LIN {X 0,Y 186.712,Z 737.862,A -85,B 0,C 180,E1 -23388.136,E2 -23388.136} C_VEL
LIN {X 0,Y 190.106,Z 731.981,A -85,B 0,C 180,E1 -23389.886,E2 -23389.886} C_VEL
LIN {X 0,Y 190.908,Z 730.143,A -85,B 0,C 180,E1 -23390.464,E2 -23390.464} C_VEL
LIN {X 0,Y 192.112,Z 723.011,A -85,B 0,C 180,E1 -23393.119,E2 -23393.119} C_VEL
LIN {X 0,Y 192.536,Z 714.54,A -85,B 0,C 180,E1 -23396.337,E2 -23396.337} C_VEL
LIN {X 0,Y 192.019,Z 709.698,A -85,B 0,C 180,E1 -23398.427,E2 -23398.427} C_VEL
LIN {X 0,Y 189.959,Z 701.617,A -85,B 0,C 180,E1 -23402.676,E2 -23402.676} C_VEL
LIN {X 0,Y 188.484,Z 698.004,A -85,B 0,C 180,E1 -23405.153,E2 -23405.153} C_VEL
LIN {X 0,Y 186.546,Z 693.819,A -85,B 0,C 180,E1 -23408.667,E2 -23408.667} C_VEL
LIN {X 0,Y 184.642,Z 689.744,A -85,B 0,C 180,E1 -23413.201,E2 -23413.201} C_VEL
LIN {X 0,Y 183.126,Z 688.308,A -85,B 0,C 180,E1 -23417.88,E2 -23417.88} C_VEL
LIN {X 0,Y 182.793,Z 688.035,A -85,B 0,C 180,E1 -23422.672,E2 -23422.672} C_VEL
LIN {X 0,Y 183.551,Z 689.151,A -85,B 0,C 180,E1 -23427.353,E2 -23427.353} C_VEL
LIN {X 0,Y 184.381,Z 690.199,A -85,B 0,C 180,E1 -23429.704,E2 -23429.704} C_VEL
LIN {X 0,Y 185.28,Z 692.119,A -85,B 0,C 180,E1 -23432.076,E2 -23432.076} C_VEL
LIN {X 0,Y 186.909,Z 695.318,A -85,B 0,C 180,E1 -23435.291,E2 -23435.291} C_VEL
LIN {X 0,Y 189.282,Z 700.42,A -85,B 0,C 180,E1 -23439.139,E2 -23439.139} C_VEL
LIN {X 0,Y 191.326,Z 707.048,A -85,B 0,C 180,E1 -23442.723,E2 -23442.723} C_VEL
LIN {X 0,Y 192.053,Z 709.901,A -85,B 0,C 180,E1 -23444.05,E2 -23444.05} C_VEL
LIN {X 0,Y 192.147,Z 713.982,A -85,B 0,C 180,E1 -23445.498,E2 -23445.498} C_VEL
LIN {X 0,Y 191.189,Z 723.676,A -85,B 0,C 180,E1 -23448.574,E2 -23448.574} C_VEL
LIN {X 0,Y 189.395,Z 732.577,A -85,B 0,C 180,E1 -23451.427,E2 -23451.427} C_VEL
LIN {X 0,Y 186.775,Z 741.156,A -85,B 0,C 180,E1 -23454.323,E2 -23454.323} C_VEL
LIN {X 0,Y 184.598,Z 745.61,A -85,B 0,C 180,E1 -23455.838,E2 -23455.838} C_VEL
LIN {X 0,Y 179.665,Z 753.449,A -85,B 0,C 180,E1 -23458.783,E2 -23458.783} C_VEL
LIN {X 0,Y 174.569,Z 760.74,A -85,B 0,C 180,E1 -23462.338,E2 -23462.338} C_VEL
LIN {X 0,Y 170.932,Z 765.844,A -85,B 0,C 180,E1 -23465.724,E2 -23465.724} C_VEL
LIN {X 0,Y 167.819,Z 769.773,A -85,B 0,C 180,E1 -23469.148,E2 -23469.148} C_VEL
LIN {X 0,Y 165.259,Z 772.729,A -85,B 0,C 180,E1 -23472.682,E2 -23472.682} C_VEL
LIN {X 0,Y 163.137,Z 775.246,A -85,B 0,C 180,E1 -23477.562,E2 -23477.562} C_VEL
LIN {X 0,Y 162.025,Z 776.252,A -85,B 0,C 180,E1 -23482.524,E2 -23482.524} C_VEL
LIN {X 0,Y 161.851,Z 775.794,A -85,B 0,C 180,E1 -23487.106,E2 -23487.106} C_VEL
LIN {X 0,Y 161.904,Z 775.442,A -85,B 0,C 180,E1 -23488.77,E2 -23488.77} C_VEL
LIN {X 0,Y 162.003,Z 776.041,A -85,B 0,C 180,E1 -23490.001,E2 -23490.001} C_VEL
LIN {X 0,Y 161.833,Z 777.013,A -85,B 0,C 180,E1 -23492.77,E2 -23492.77} C_VEL
LIN {X 0,Y 162.035,Z 777.558,A -85,B 0,C 180,E1 -23497.478,E2 -23497.478} C_VEL
LIN {X 0,Y 163.149,Z 776.604,A -85,B 0,C 180,E1 -23502.439,E2 -23502.439} C_VEL
LIN {X 0,Y 163.38,Z 776.322,A -85,B 0,C 180,E1 -23503.114,E2 -23503.114} C_VEL
LIN {X 0,Y 163.558,Z 775.484,A -85,B 0,C 180,E1 -23505.161,E2 -23505.161} C_VEL
LIN {X 0,Y 162.556,Z 773.609,A -85,B 0,C 180,E1 -23508.569,E2 -23508.569} C_VEL
LIN {X 0,Y 162.155,Z 771.222,A -85,B 0,C 180,E1 -23511.955,E2 -23511.955} C_VEL
LIN {X 0,Y 163.246,Z 769.393,A -85,B 0,C 180,E1 -23513.891,E2 -23513.891} C_VEL
LIN {X 0,Y 167.46,Z 764.248,A -85,B 0,C 180,E1 -23517.989,E2 -23517.989} C_VEL
LIN {X 0,Y 172.073,Z 758.395,A -85,B 0,C 180,E1 -23521.384,E2 -23521.384} C_VEL
LIN {X 0,Y 177.108,Z 751.485,A -85,B 0,C 180,E1 -23524.436,E2 -23524.436} C_VEL
LIN {X 0,Y 180.696,Z 746.067,A -85,B 0,C 180,E1 -23526.381,E2 -23526.381} C_VEL
LIN {X 0,Y 183.191,Z 739.813,A -85,B 0,C 180,E1 -23528.764,E2 -23528.764} C_VEL
LIN {X 0,Y 185.082,Z 732.261,A -85,B 0,C 180,E1 -23531.646,E2 -23531.646} C_VEL
LIN {X 0,Y 186.028,Z 725.848,A -85,B 0,C 180,E1 -23534.126,E2 -23534.126} C_VEL
LIN {X 0,Y 186.099,Z 721.842,A -85,B 0,C 180,E1 -23535.852,E2 -23535.852} C_VEL
LIN {X 0,Y 185.417,Z 716.956,A -85,B 0,C 180,E1 -23538.448,E2 -23538.448} C_VEL
LIN {X 0,Y 183.96,Z 710.944,A -85,B 0,C 180,E1 -23542.319,E2 -23542.319} C_VEL
LIN {X 0,Y 183.024,Z 707.744,A -85,B 0,C 180,E1 -23544.831,E2 -23544.831} C_VEL
LIN {X 0,Y 181.454,Z 703.142,A -85,B 0,C 180,E1 -23549.767,E2 -23549.767} C_VEL
LIN {X 0,Y 181.071,Z 701.312,A -85,B 0,C 180,E1 -23552.24,E2 -23552.24} C_VEL
LIN {X 0,Y 180.413,Z 699.995,A -85,B 0,C 180,E1 -23557.074,E2 -23557.074} C_VEL
LIN {X 0,Y 180.881,Z 699.879,A -85,B 0,C 180,E1 -23561.891,E2 -23561.891} C_VEL
LIN {X 0,Y 181.587,Z 700.232,A -85,B 0,C 180,E1 -23564.281,E2 -23564.281} C_VEL
LIN {X 0,Y 182.735,Z 703.422,A -85,B 0,C 180,E1 -23568.913,E2 -23568.913} C_VEL
LIN {X 0,Y 183.638,Z 705.359,A -85,B 0,C 180,E1 -23571.194,E2 -23571.194} C_VEL
LIN {X 0,Y 185.128,Z 709.014,A -85,B 0,C 180,E1 -23574.554,E2 -23574.554} C_VEL
LIN {X 0,Y 186.172,Z 712.751,A -85,B 0,C 180,E1 -23577.188,E2 -23577.188} C_VEL
LIN {X 0,Y 187.119,Z 718.537,A -85,B 0,C 180,E1 -23580.538,E2 -23580.538} C_VEL
LIN {X 0,Y 187.078,Z 723.111,A -85,B 0,C 180,E1 -23582.692,E2 -23582.692} C_VEL
LIN {X 0,Y 186.215,Z 730.51,A -85,B 0,C 180,E1 -23585.957,E2 -23585.957} C_VEL
LIN {X 0,Y 185.472,Z 733.89,A -85,B 0,C 180,E1 -23587.406,E2 -23587.406} C_VEL
LIN {X 0,Y 182.996,Z 738.287,A -85,B 0,C 180,E1 -23588.837,E2 -23588.837} C_VEL
LIN {X 0,Y 177.113,Z 746.781,A -85,B 0,C 180,E1 -23592.017,E2 -23592.017} C_VEL
LIN {X 0,Y 171.766,Z 753.637,A -85,B 0,C 180,E1 -23595.424,E2 -23595.424} C_VEL
LIN {X 0,Y 167.943,Z 758.159,A -85,B 0,C 180,E1 -23598.405,E2 -23598.405} C_VEL
LIN {X 0,Y 164.43,Z 761.942,A -85,B 0,C 180,E1 -23601.652,E2 -23601.652} C_VEL
LIN {X 0,Y 160.739,Z 765.467,A -85,B 0,C 180,E1 -23605.927,E2 -23605.927} C_VEL
LIN {X 0,Y 158.579,Z 767.219,A -85,B 0,C 180,E1 -23609.177,E2 -23609.177} C_VEL
LIN {X 0,Y 156.907,Z 768.33,A -85,B 0,C 180,E1 -23612.513,E2 -23612.513} C_VEL
LIN {X 0,Y 155.638,Z 768.732,A -85,B 0,C 180,E1 -23615.947,E2 -23615.947} C_VEL
LIN {X 0,Y 154.834,Z 768.465,A -85,B 0,C 180,E1 -23619.497,E2 -23619.497} C_VEL
LIN {X 0,Y 154.381,Z 767.416,A -85,B 0,C 180,E1 -23623.248,E2 -23623.248} C_VEL
LIN {X 0,Y 154.361,Z 765.565,A -85,B 0,C 180,E1 -23626.925,E2 -23626.925} C_VEL
LIN {X 0,Y 154.778,Z 762.954,A -85,B 0,C 180,E1 -23630.527,E2 -23630.527} C_VEL
LIN {X 0,Y 155.489,Z 759.109,A -85,B 0,C 180,E1 -23634.448,E2 -23634.448} C_VEL
LIN {X 0,Y 156.66,Z 753.93,A -85,B 0,C 180,E1 -23638.471,E2 -23638.471} C_VEL
LIN {X 0,Y 158.448,Z 747.231,A -85,B 0,C 180,E1 -23642.512,E2 -23642.512} C_VEL
LIN {X 0,Y 160.896,Z 738.567,A -85,B 0,C 180,E1 -23646.533,E2 -23646.533} C_VEL
LIN {X 0,Y 163.527,Z 729.361,A -85,B 0,C 180,E1 -23649.889,E2 -23649.889} C_VEL
LIN {X 0,Y 166.295,Z 719.218,A -85,B 0,C 180,E1 -23652.791,E2 -23652.791} C_VEL
LIN {X 0,Y 167.408,Z 714.851,A -85,B 0,C 180,E1 -23653.851,E2 -23653.851} C_VEL
LIN {X 0,Y 166.812,Z 706.424,A -85,B 0,C 180,E1 -23655.978,E2 -23655.978} C_VEL
LIN {X 0,Y 165.34,Z 695.499,A -85,B 0,C 180,E1 -23658.413,E2 -23658.413} C_VEL
LIN {X 0,Y 163.12,Z 683.74,A -85,B 0,C 180,E1 -23660.701,E2 -23660.701} C_VEL
LIN {X 0,Y 159.913,Z 670.534,A -85,B 0,C 180,E1 -23662.899,E2 -23662.899} C_VEL
LIN {X 0,Y 158.501,Z 667.234,A -85,B 0,C 180,E1 -23663.475,E2 -23663.475} C_VEL
LIN {X 0,Y 157.726,Z 664.838,A -85,B 0,C 180,E1 -23663.924,E2 -23663.924} C_VEL
LIN {X 0,Y 158.258,Z 664.771,A -85,B 0,C 180,E1 -23669.999,E2 -23669.999} C_VEL
LIN {X 0,Y 157.677,Z 664.846,A -85,B 0,C 180,E1 -23675.354,E2 -23675.354} C_VEL
LIN {X 0,Y 158.763,Z 667.875,A -85,B 0,C 180,E1 -23675.874,E2 -23675.874} C_VEL
LIN {X 0,Y 162.128,Z 676.352,A -85,B 0,C 180,E1 -23677.393,E2 -23677.393} C_VEL
LIN {X 0,Y 164.537,Z 688.841,A -85,B 0,C 180,E1 -23679.554,E2 -23679.554} C_VEL
LIN {X 0,Y 166.157,Z 699.914,A -85,B 0,C 180,E1 -23681.804,E2 -23681.804} C_VEL
LIN {X 0,Y 167.206,Z 710.54,A -85,B 0,C 180,E1 -23684.295,E2 -23684.295} C_VEL
LIN {X 0,Y 167.459,Z 713.795,A -85,B 0,C 180,E1 -23685.143,E2 -23685.143} C_VEL
LIN {X 0,Y 164.601,Z 724.758,A -85,B 0,C 180,E1 -23687.961,E2 -23687.961} C_VEL
LIN {X 0,Y 162.062,Z 733.921,A -85,B 0,C 180,E1 -23690.962,E2 -23690.962} C_VEL
LIN {X 0,Y 159.416,Z 743.059,A -85,B 0,C 180,E1 -23694.759,E2 -23694.759} C_VEL
LIN {X 0,Y 157.616,Z 749.693,A -85,B 0,C 180,E1 -23698.256,E2 -23698.256} C_VEL
LIN {X 0,Y 156.377,Z 754.45,A -85,B 0,C 180,E1 -23701.36,E2 -23701.36} C_VEL
LIN {X 0,Y 155.235,Z 759.42,A -85,B 0,C 180,E1 -23705.42,E2 -23705.42} C_VEL
LIN {X 0,Y 154.449,Z 763.205,A -85,B 0,C 180,E1 -23709.571,E2 -23709.571} C_VEL
LIN {X 0,Y 154.222,Z 765.534,A -85,B 0,C 180,E1 -23713.186,E2 -23713.186} C_VEL
LIN {X 0,Y 154.357,Z 767.123,A -85,B 0,C 180,E1 -23716.924,E2 -23716.924} C_VEL
LIN {X 0,Y 154.91,Z 767.907,A -85,B 0,C 180,E1 -23720.568,E2 -23720.568} C_VEL
LIN {X 0,Y 155.925,Z 767.942,A -85,B 0,C 180,E1 -23724.222,E2 -23724.222} C_VEL
LIN {X 0,Y 157.494,Z 767.132,A -85,B 0,C 180,E1 -23727.976,E2 -23727.976} C_VEL
LIN {X 0,Y 159.633,Z 765.454,A -85,B 0,C 180,E1 -23731.702,E2 -23731.702} C_VEL
LIN {X 0,Y 162.394,Z 762.886,A -85,B 0,C 180,E1 -23735.341,E2 -23735.341} C_VEL
LIN {X 0,Y 165.753,Z 759.343,A -85,B 0,C 180,E1 -23738.874,E2 -23738.874} C_VEL
LIN {X 0,Y 169.733,Z 754.752,A -85,B 0,C 180,E1 -23742.235,E2 -23742.235} C_VEL
LIN {X 0,Y 174.266,Z 748.995,A -85,B 0,C 180,E1 -23745.438,E2 -23745.438} C_VEL
LIN {X 0,Y 179.772,Z 741.207,A -85,B 0,C 180,E1 -23748.728,E2 -23748.728} C_VEL
LIN {X 0,Y 184.839,Z 733.12,A -85,B 0,C 180,E1 -23751.323,E2 -23751.323} C_VEL
LIN {X 0,Y 185.992,Z 729.01,A -85,B 0,C 180,E1 -23752.913,E2 -23752.913} C_VEL
LIN {X 0,Y 187.104,Z 722.14,A -85,B 0,C 180,E1 -23755.692,E2 -23755.692} C_VEL
LIN {X 0,Y 187.392,Z 716.951,A -85,B 0,C 180,E1 -23757.851,E2 -23757.851} C_VEL
LIN {X 0,Y 186.623,Z 711.316,A -85,B 0,C 180,E1 -23760.783,E2 -23760.783} C_VEL
LIN {X 0,Y 185.786,Z 707.026,A -85,B 0,C 180,E1 -23763.253,E2 -23763.253} C_VEL
LIN {X 0,Y 184.533,Z 703.526,A -85,B 0,C 180,E1 -23765.839,E2 -23765.839} C_VEL
LIN {X 0,Y 183.23,Z 700.177,A -85,B 0,C 180,E1 -23768.825,E2 -23768.825} C_VEL
LIN {X 0,Y 181.68,Z 696.213,A -85,B 0,C 180,E1 -23773.421,E2 -23773.421} C_VEL
LIN {X 0,Y 180.353,Z 694.814,A -85,B 0,C 180,E1 -23778.164,E2 -23778.164} C_VEL
LIN {X 0,Y 180.118,Z 694.644,A -85,B 0,C 180,E1 -23782.966,E2 -23782.966} C_VEL
LIN {X 0,Y 180.917,Z 695.911,A -85,B 0,C 180,E1 -23787.785,E2 -23787.785} C_VEL
LIN {X 0,Y 181.693,Z 697.21,A -85,B 0,C 180,E1 -23790.189,E2 -23790.189} C_VEL
LIN {X 0,Y 183.599,Z 701.621,A -85,B 0,C 180,E1 -23795.043,E2 -23795.043} C_VEL
LIN {X 0,Y 185.399,Z 706.086,A -85,B 0,C 180,E1 -23798.583,E2 -23798.583} C_VEL
LIN {X 0,Y 187.123,Z 713.019,A -85,B 0,C 180,E1 -23802.536,E2 -23802.536} C_VEL
LIN {X 0,Y 187.343,Z 716.031,A -85,B 0,C 180,E1 -23803.859,E2 -23803.859} C_VEL
LIN {X 0,Y 186.21,Z 724.617,A -85,B 0,C 180,E1 -23806.804,E2 -23806.804} C_VEL
LIN {X 0,Y 184.276,Z 733.14,A -85,B 0,C 180,E1 -23809.709,E2 -23809.709} C_VEL
LIN {X 0,Y 181.73,Z 740.888,A -85,B 0,C 180,E1 -23812.477,E2 -23812.477} C_VEL
LIN {X 0,Y 179.722,Z 745.256,A -85,B 0,C 180,E1 -23814.087,E2 -23814.087} C_VEL
LIN {X 0,Y 174.506,Z 753.117,A -85,B 0,C 180,E1 -23817.066,E2 -23817.066} C_VEL
LIN {X 0,Y 169.726,Z 759.549,A -85,B 0,C 180,E1 -23820.207,E2 -23820.207} C_VEL
LIN {X 0,Y 165.66,Z 764.734,A -85,B 0,C 180,E1 -23823.549,E2 -23823.549} C_VEL
LIN {X 0,Y 162.274,Z 768.848,A -85,B 0,C 180,E1 -23827.06,E2 -23827.06} C_VEL
LIN {X 0,Y 160.211,Z 771.067,A -85,B 0,C 180,E1 -23829.457,E2 -23829.457} C_VEL
LIN {X 0,Y 158.477,Z 772.835,A -85,B 0,C 180,E1 -23831.916,E2 -23831.916} C_VEL
LIN {X 0,Y 156.187,Z 775.195,A -85,B 0,C 180,E1 -23836.999,E2 -23836.999} C_VEL
LIN {X 0,Y 155.443,Z 775.823,A -85,B 0,C 180,E1 -23839.582,E2 -23839.582} C_VEL
LIN {X 0,Y 154.971,Z 776.051,A -85,B 0,C 180,E1 -23842.182,E2 -23842.182} C_VEL
LIN {X 0,Y 154.783,Z 775.877,A -85,B 0,C 180,E1 -23844.791,E2 -23844.791} C_VEL
LIN {X 0,Y 154.831,Z 774.955,A -85,B 0,C 180,E1 -23848.697,E2 -23848.697} C_VEL
LIN {X 0,Y 154.91,Z 775.623,A -85,B 0,C 180,E1 -23850.001,E2 -23850.001} C_VEL
LIN {X 0,Y 154.746,Z 776.569,A -85,B 0,C 180,E1 -23852.604,E2 -23852.604} C_VEL
LIN {X 0,Y 154.781,Z 777.133,A -85,B 0,C 180,E1 -23855.211,E2 -23855.211} C_VEL
LIN {X 0,Y 155.456,Z 777.136,A -85,B 0,C 180,E1 -23860.42,E2 -23860.42} C_VEL
LIN {X 0,Y 157.208,Z 775.581,A -85,B 0,C 180,E1 -23865.56,E2 -23865.56} C_VEL
LIN {X 0,Y 160.266,Z 772.531,A -85,B 0,C 180,E1 -23870.538,E2 -23870.538} C_VEL
LIN {X 0,Y 163.246,Z 769.393,A -85,B 0,C 180,E1 -23873.891,E2 -23873.891} C_VEL
LIN {X 0,Y 163.829,Z 768.103,A -85,B 0,C 180,E1 -23875.198,E2 -23875.198} C_VEL
LIN {X 0,Y 163.133,Z 766.066,A -85,B 0,C 180,E1 -23877.448,E2 -23877.448} C_VEL
LIN {X 0,Y 162.649,Z 763.801,A -85,B 0,C 180,E1 -23879.682,E2 -23879.682} C_VEL
LIN {X 0,Y 163.534,Z 762.125,A -85,B 0,C 180,E1 -23880.914,E2 -23880.914} C_VEL
LIN {X 0,Y 168.641,Z 755.959,A -85,B 0,C 180,E1 -23884.237,E2 -23884.237} C_VEL
LIN {X 0,Y 174.162,Z 748.613,A -85,B 0,C 180,E1 -23887.251,E2 -23887.251} C_VEL
LIN {X 0,Y 175.79,Z 745.856,A -85,B 0,C 180,E1 -23888.294,E2 -23888.294} C_VEL
LIN {X 0,Y 178.272,Z 739.539,A -85,B 0,C 180,E1 -23890.899,E2 -23890.899} C_VEL
LIN {X 0,Y 180.181,Z 732.465,A -85,B 0,C 180,E1 -23893.817,E2 -23893.817} C_VEL
LIN {X 0,Y 180.864,Z 728.249,A -85,B 0,C 180,E1 -23895.618,E2 -23895.618} C_VEL
LIN {X 0,Y 180.912,Z 724.418,A -85,B 0,C 180,E1 -23897.571,E2 -23897.571} C_VEL
LIN {X 0,Y 180.434,Z 720.331,A -85,B 0,C 180,E1 -23900.009,E2 -23900.009} C_VEL
LIN {X 0,Y 179.734,Z 716.555,A -85,B 0,C 180,E1 -23902.702,E2 -23902.702} C_VEL
LIN {X 0,Y 178.671,Z 712.164,A -85,B 0,C 180,E1 -23906.586,E2 -23906.586} C_VEL
LIN {X 0,Y 177.698,Z 708.058,A -85,B 0,C 180,E1 -23911.667,E2 -23911.667} C_VEL
LIN {X 0,Y 177.351,Z 706.922,A -85,B 0,C 180,E1 -23914.157,E2 -23914.157} C_VEL
LIN {X 0,Y 177.183,Z 706.121,A -85,B 0,C 180,E1 -23919.085,E2 -23919.085} C_VEL
LIN {X 0,Y 178.103,Z 706.432,A -85,B 0,C 180,E1 -23923.965,E2 -23923.965} C_VEL
LIN {X 0,Y 179.061,Z 709.599,A -85,B 0,C 180,E1 -23928.884,E2 -23928.884} C_VEL
LIN {X 0,Y 180.21,Z 712.8,A -85,B 0,C 180,E1 -23932.516,E2 -23932.516} C_VEL
LIN {X 0,Y 181.234,Z 716.246,A -85,B 0,C 180,E1 -23935.552,E2 -23935.552} C_VEL
LIN {X 0,Y 181.903,Z 721.342,A -85,B 0,C 180,E1 -23938.893,E2 -23938.893} C_VEL
LIN {X 0,Y 181.891,Z 725.332,A -85,B 0,C 180,E1 -23941.107,E2 -23941.107} C_VEL
LIN {X 0,Y 180.818,Z 732.308,A -85,B 0,C 180,E1 -23944.459,E2 -23944.459} C_VEL
LIN {X 0,Y 179.859,Z 735.959,A -85,B 0,C 180,E1 -23946.169,E2 -23946.169} C_VEL
LIN {X 0,Y 175.815,Z 742.199,A -85,B 0,C 180,E1 -23948.322,E2 -23948.322} C_VEL
LIN {X 0,Y 170.597,Z 749.046,A -85,B 0,C 180,E1 -23951.171,E2 -23951.171} C_VEL
LIN {X 0,Y 164.883,Z 755.647,A -85,B 0,C 180,E1 -23954.818,E2 -23954.818} C_VEL
LIN {X 0,Y 161.094,Z 759.676,A -85,B 0,C 180,E1 -23957.782,E2 -23957.782} C_VEL
LIN {X 0,Y 156.181,Z 764.286,A -85,B 0,C 180,E1 -23962.488,E2 -23962.488} C_VEL
LIN {X 0,Y 152.389,Z 767.295,A -85,B 0,C 180,E1 -23967.464,E2 -23967.464} C_VEL
LIN {X 0,Y 149.789,Z 768.73,A -85,B 0,C 180,E1 -23972.375,E2 -23972.375} C_VEL
LIN {X 0,Y 147.973,Z 768.797,A -85,B 0,C 180,E1 -23978.129,E2 -23978.129} C_VEL
LIN {X 0,Y 147.393,Z 767.88,A -85,B 0,C 180,E1 -23981.879,E2 -23981.879} C_VEL
LIN {X 0,Y 147.228,Z 766.194,A -85,B 0,C 180,E1 -23985.728,E2 -23985.728} C_VEL
LIN {X 0,Y 147.553,Z 763.649,A -85,B 0,C 180,E1 -23989.649,E2 -23989.649} C_VEL
LIN {X 0,Y 148.227,Z 760.03,A -85,B 0,C 180,E1 -23993.711,E2 -23993.711} C_VEL
LIN {X 0,Y 149.324,Z 755.089,A -85,B 0,C 180,E1 -23997.907,E2 -23997.907} C_VEL
LIN {X 0,Y 151.082,Z 748.412,A -85,B 0,C 180,E1 -24002.277,E2 -24002.277} C_VEL
LIN {X 0,Y 153.473,Z 740.442,A -85,B 0,C 180,E1 -24006.329,E2 -24006.329} C_VEL
LIN {X 0,Y 155.942,Z 731.984,A -85,B 0,C 180,E1 -24009.701,E2 -24009.701} C_VEL
LIN {X 0,Y 158.943,Z 721.609,A -85,B 0,C 180,E1 -24012.966,E2 -24012.966} C_VEL
LIN {X 0,Y 160.628,Z 714.624,A -85,B 0,C 180,E1 -24014.779,E2 -24014.779} C_VEL
LIN {X 0,Y 159.59,Z 703.661,A -85,B 0,C 180,E1 -24017.634,E2 -24017.634} C_VEL
LIN {X 0,Y 158.012,Z 692.808,A -85,B 0,C 180,E1 -24020.075,E2 -24020.075} C_VEL
LIN {X 0,Y 155.855,Z 681.966,A -85,B 0,C 180,E1 -24022.224,E2 -24022.224} C_VEL
LIN {X 0,Y 153.244,Z 671.76,A -85,B 0,C 180,E1 -24024.035,E2 -24024.035} C_VEL
LIN {X 0,Y 150.838,Z 666.576,A -85,B 0,C 180,E1 -24025.071,E2 -24025.071} C_VEL
LIN {X 0,Y 150.7,Z 665.712,A -85,B 0,C 180,E1 -24025.318,E2 -24025.318} C_VEL
LIN {X 0,Y 151.218,Z 665.648,A -85,B 0,C 180,E1 -24029.999,E2 -24029.999} C_VEL
LIN {X 0,Y 150.738,Z 665.905,A -85,B 0,C 180,E1 -24034.093,E2 -24034.093} C_VEL
LIN {X 0,Y 151.813,Z 668.79,A -85,B 0,C 180,E1 -24034.604,E2 -24034.604} C_VEL
LIN {X 0,Y 155.865,Z 678.865,A -85,B 0,C 180,E1 -24036.595,E2 -24036.595} C_VEL
LIN {X 0,Y 158.207,Z 691.938,A -85,B 0,C 180,E1 -24039.049,E2 -24039.049} C_VEL
LIN {X 0,Y 159.66,Z 702.785,A -85,B 0,C 180,E1 -24041.424,E2 -24041.424} C_VEL
LIN {X 0,Y 160.566,Z 713.802,A -85,B 0,C 180,E1 -24044.252,E2 -24044.252} C_VEL
LIN {X 0,Y 159.327,Z 719.367,A -85,B 0,C 180,E1 -24045.674,E2 -24045.674} C_VEL
LIN {X 0,Y 156.522,Z 729.436,A -85,B 0,C 180,E1 -24048.688,E2 -24048.688} C_VEL
LIN {X 0,Y 153.859,Z 738.321,A -85,B 0,C 180,E1 -24052.069,E2 -24052.069} C_VEL
LIN {X 0,Y 151.448,Z 746.582,A -85,B 0,C 180,E1 -24056.073,E2 -24056.073} C_VEL
LIN {X 0,Y 149.589,Z 753.402,A -85,B 0,C 180,E1 -24060.334,E2 -24060.334} C_VEL
LIN {X 0,Y 148.276,Z 758.714,A -85,B 0,C 180,E1 -24064.663,E2 -24064.663} C_VEL
LIN {X 0,Y 147.544,Z 762.128,A -85,B 0,C 180,E1 -24068.258,E2 -24068.258} C_VEL
LIN {X 0,Y 147.155,Z 764.792,A -85,B 0,C 180,E1 -24071.96,E2 -24071.96} C_VEL
LIN {X 0,Y 147.167,Z 766.685,A -85,B 0,C 180,E1 -24075.75,E2 -24075.75} C_VEL
LIN {X 0,Y 147.609,Z 767.842,A -85,B 0,C 180,E1 -24079.621,E2 -24079.621} C_VEL
LIN {X 0,Y 148.545,Z 768.228,A -85,B 0,C 180,E1 -24083.541,E2 -24083.541} C_VEL
LIN {X 0,Y 150.064,Z 767.811,A -85,B 0,C 180,E1 -24087.456,E2 -24087.456} C_VEL
LIN {X 0,Y 152.986,Z 765.888,A -85,B 0,C 180,E1 -24092.652,E2 -24092.652} C_VEL
LIN {X 0,Y 156.974,Z 762.504,A -85,B 0,C 180,E1 -24097.553,E2 -24097.553} C_VEL
LIN {X 0,Y 160.383,Z 759.155,A -85,B 0,C 180,E1 -24100.813,E2 -24100.813} C_VEL
LIN {X 0,Y 165.186,Z 753.943,A -85,B 0,C 180,E1 -24104.579,E2 -24104.579} C_VEL
LIN {X 0,Y 170.697,Z 747.199,A -85,B 0,C 180,E1 -24108.12,E2 -24108.12} C_VEL
LIN {X 0,Y 176.788,Z 738.848,A -85,B 0,C 180,E1 -24111.387,E2 -24111.387} C_VEL
LIN {X 0,Y 179.162,Z 735.261,A -85,B 0,C 180,E1 -24112.534,E2 -24112.534} C_VEL
LIN {X 0,Y 180.694,Z 730.715,A -85,B 0,C 180,E1 -24114.42,E2 -24114.42} C_VEL
LIN {X 0,Y 182.125,Z 723.016,A -85,B 0,C 180,E1 -24117.788,E2 -24117.788} C_VEL
LIN {X 0,Y 182.269,Z 719.618,A -85,B 0,C 180,E1 -24119.448,E2 -24119.448} C_VEL
LIN {X 0,Y 181.493,Z 713.117,A -85,B 0,C 180,E1 -24123.33,E2 -24123.33} C_VEL
LIN {X 0,Y 181.206,Z 711.44,A -85,B 0,C 180,E1 -24124.449,E2 -24124.449} C_VEL
LIN {X 0,Y 179.582,Z 706.307,A -85,B 0,C 180,E1 -24129.006,E2 -24129.006} C_VEL
LIN {X 0,Y 178.367,Z 702.486,A -85,B 0,C 180,E1 -24133.675,E2 -24133.675} C_VEL
LIN {X 0,Y 177.249,Z 701.19,A -85,B 0,C 180,E1 -24138.494,E2 -24138.494} C_VEL
LIN {X 0,Y 177.115,Z 701.141,A -85,B 0,C 180,E1 -24143.379,E2 -24143.379} C_VEL
LIN {X 0,Y 177.425,Z 701.664,A -85,B 0,C 180,E1 -24145.831,E2 -24145.831} C_VEL
LIN {X 0,Y 178.435,Z 703.477,A -85,B 0,C 180,E1 -24149.947,E2 -24149.947} C_VEL
LIN {X 0,Y 180.047,Z 707.893,A -85,B 0,C 180,E1 -24154.946,E2 -24154.946} C_VEL
LIN {X 0,Y 181.359,Z 712.066,A -85,B 0,C 180,E1 -24158.318,E2 -24158.318} C_VEL
LIN {X 0,Y 182.374,Z 717.42,A -85,B 0,C 180,E1 -24161.588,E2 -24161.588} C_VEL
LIN {X 0,Y 182.406,Z 720.274,A -85,B 0,C 180,E1 -24162.942,E2 -24162.942} C_VEL
LIN {X 0,Y 180.99,Z 727.677,A -85,B 0,C 180,E1 -24165.658,E2 -24165.658} C_VEL
LIN {X 0,Y 178.713,Z 735.575,A -85,B 0,C 180,E1 -24168.559,E2 -24168.559} C_VEL
LIN {X 0,Y 175.551,Z 743.638,A -85,B 0,C 180,E1 -24171.647,E2 -24171.647} C_VEL
LIN {X 0,Y 173.162,Z 747.8,A -85,B 0,C 180,E1 -24173.228,E2 -24173.228} C_VEL
LIN {X 0,Y 167.796,Z 755.107,A -85,B 0,C 180,E1 -24176.293,E2 -24176.293} C_VEL
LIN {X 0,Y 161.787,Z 762.349,A -85,B 0,C 180,E1 -24180.319,E2 -24180.319} C_VEL
LIN {X 0,Y 158.077,Z 766.631,A -85,B 0,C 180,E1 -24183.604,E2 -24183.604} C_VEL
LIN {X 0,Y 154.63,Z 770.245,A -85,B 0,C 180,E1 -24187.275,E2 -24187.275} C_VEL
LIN {X 0,Y 151.731,Z 772.928,A -85,B 0,C 180,E1 -24191.082,E2 -24191.082} C_VEL
LIN {X 0,Y 149.239,Z 775.157,A -85,B 0,C 180,E1 -24196.382,E2 -24196.382} C_VEL
LIN {X 0,Y 147.94,Z 775.818,A -85,B 0,C 180,E1 -24201.808,E2 -24201.808} C_VEL
LIN {X 0,Y 147.695,Z 774.975,A -85,B 0,C 180,E1 -24207.274,E2 -24207.274} C_VEL
LIN {X 0,Y 147.763,Z 774.546,A -85,B 0,C 180,E1 -24208.808,E2 -24208.808} C_VEL
LIN {X 0,Y 147.689,Z 775.991,A -85,B 0,C 180,E1 -24212.114,E2 -24212.114} C_VEL
LIN {X 0,Y 147.704,Z 776.82,A -85,B 0,C 180,E1 -24215.462,E2 -24215.462} C_VEL
LIN {X 0,Y 148.474,Z 776.957,A -85,B 0,C 180,E1 -24220.915,E2 -24220.915} C_VEL
LIN {X 0,Y 150.343,Z 775.6,A -85,B 0,C 180,E1 -24226.29,E2 -24226.29} C_VEL
LIN {X 0,Y 153.627,Z 772.703,A -85,B 0,C 180,E1 -24231.469,E2 -24231.469} C_VEL
LIN {X 0,Y 157.02,Z 769.483,A -85,B 0,C 180,E1 -24235.165,E2 -24235.165} C_VEL
LIN {X 0,Y 162.173,Z 763.695,A -85,B 0,C 180,E1 -24239.919,E2 -24239.919} C_VEL
LIN {X 0,Y 163.534,Z 762.125,A -85,B 0,C 180,E1 -24240.914,E2 -24240.914} C_VEL
LIN {X 0,Y 165.453,Z 759.45,A -85,B 0,C 180,E1 -24242.621,E2 -24242.621} C_VEL
LIN {X 0,Y 167.438,Z 754.846,A -85,B 0,C 180,E1 -24245.549,E2 -24245.549} C_VEL
LIN {X 0,Y 168.756,Z 750.884,A -85,B 0,C 180,E1 -24247.866,E2 -24247.866} C_VEL
LIN {X 0,Y 170.587,Z 746.519,A -85,B 0,C 180,E1 -24250.028,E2 -24250.028} C_VEL
LIN {X 0,Y 172.893,Z 741.185,A -85,B 0,C 180,E1 -24252.4,E2 -24252.4} C_VEL
LIN {X 0,Y 175.059,Z 734.335,A -85,B 0,C 180,E1 -24255.431,E2 -24255.431} C_VEL
LIN {X 0,Y 175.762,Z 730.746,A -85,B 0,C 180,E1 -24257.175,E2 -24257.175} C_VEL
LIN {X 0,Y 175.688,Z 725.805,A -85,B 0,C 180,E1 -24260.205,E2 -24260.205} C_VEL
LIN {X 0,Y 175.189,Z 721.65,A -85,B 0,C 180,E1 -24263.354,E2 -24263.354} C_VEL
LIN {X 0,Y 174.744,Z 719.011,A -85,B 0,C 180,E1 -24265.732,E2 -24265.732} C_VEL
LIN {X 0,Y 173.945,Z 714.649,A -85,B 0,C 180,E1 -24270.998,E2 -24270.998} C_VEL
LIN {X 0,Y 173.678,Z 713.275,A -85,B 0,C 180,E1 -24273.569,E2 -24273.569} C_VEL
LIN {X 0,Y 173.517,Z 712.575,A -85,B 0,C 180,E1 -24276.107,E2 -24276.107} C_VEL
LIN {X 0,Y 173.768,Z 712.22,A -85,B 0,C 180,E1 -24281.122,E2 -24281.122} C_VEL
LIN {X 0,Y 174.301,Z 712.413,A -85,B 0,C 180,E1 -24283.606,E2 -24283.606} C_VEL
LIN {X 0,Y 174.98,Z 715.223,A -85,B 0,C 180,E1 -24288.415,E2 -24288.415} C_VEL
LIN {X 0,Y 175.909,Z 718.432,A -85,B 0,C 180,E1 -24292.332,E2 -24292.332} C_VEL
LIN {X 0,Y 176.599,Z 721.847,A -85,B 0,C 180,E1 -24295.435,E2 -24295.435} C_VEL
LIN {X 0,Y 176.811,Z 726.824,A -85,B 0,C 180,E1 -24298.861,E2 -24298.861} C_VEL
LIN {X 0,Y 176.436,Z 729.897,A -85,B 0,C 180,E1 -24300.628,E2 -24300.628} C_VEL
LIN {X 0,Y 174.862,Z 736.468,A -85,B 0,C 180,E1 -24304.033,E2 -24304.033} C_VEL
LIN {X 0,Y 173.706,Z 739.185,A -85,B 0,C 180,E1 -24305.277,E2 -24305.277} C_VEL
LIN {X 0,Y 167.324,Z 747.411,A -85,B 0,C 180,E1 -24308.454,E2 -24308.454} C_VEL
LIN {X 0,Y 161.188,Z 754.303,A -85,B 0,C 180,E1 -24311.984,E2 -24311.984} C_VEL
LIN {X 0,Y 156.022,Z 759.534,A -85,B 0,C 180,E1 -24315.681,E2 -24315.681} C_VEL
LIN {X 0,Y 152.311,Z 762.845,A -85,B 0,C 180,E1 -24318.845,E2 -24318.845} C_VEL
LIN {X 0,Y 149.045,Z 765.445,A -85,B 0,C 180,E1 -24322.162,E2 -24322.162} C_VEL
LIN {X 0,Y 146.353,Z 767.356,A -85,B 0,C 180,E1 -24325.607,E2 -24325.607} C_VEL
LIN {X 0,Y 144.112,Z 768.576,A -85,B 0,C 180,E1 -24329.188,E2 -24329.188} C_VEL
LIN {X 0,Y 142.378,Z 769.17,A -85,B 0,C 180,E1 -24332.948,E2 -24332.948} C_VEL
LIN {X 0,Y 141.082,Z 769.029,A -85,B 0,C 180,E1 -24337.15,E2 -24337.15} C_VEL
LIN {X 0,Y 140.355,Z 768.049,A -85,B 0,C 180,E1 -24341.313,E2 -24341.313} C_VEL
LIN {X 0,Y 140.132,Z 766.304,A -85,B 0,C 180,E1 -24345.4,E2 -24345.4} C_VEL
LIN {X 0,Y 140.43,Z 763.791,A -85,B 0,C 180,E1 -24349.412,E2 -24349.412} C_VEL
LIN {X 0,Y 141.039,Z 760.553,A -85,B 0,C 180,E1 -24353.275,E2 -24353.275} C_VEL
LIN {X 0,Y 142.238,Z 755.129,A -85,B 0,C 180,E1 -24358.118,E2 -24358.118} C_VEL
LIN {X 0,Y 144.176,Z 748.062,A -85,B 0,C 180,E1 -24362.911,E2 -24362.911} C_VEL
LIN {X 0,Y 146.482,Z 740.623,A -85,B 0,C 180,E1 -24366.822,E2 -24366.822} C_VEL
LIN {X 0,Y 149.409,Z 730.991,A -85,B 0,C 180,E1 -24370.774,E2 -24370.774} C_VEL
LIN {X 0,Y 152.35,Z 721.181,A -85,B 0,C 180,E1 -24373.931,E2 -24373.931} C_VEL
LIN {X 0,Y 153.811,Z 715.69,A -85,B 0,C 180,E1 -24375.406,E2 -24375.406} C_VEL
LIN {X 0,Y 152.852,Z 704.665,A -85,B 0,C 180,E1 -24378.43,E2 -24378.43} C_VEL
LIN {X 0,Y 151.227,Z 693.157,A -85,B 0,C 180,E1 -24381.18,E2 -24381.18} C_VEL
LIN {X 0,Y 148.829,Z 680.937,A -85,B 0,C 180,E1 -24383.731,E2 -24383.731} C_VEL
LIN {X 0,Y 147.207,Z 674.897,A -85,B 0,C 180,E1 -24384.906,E2 -24384.906} C_VEL
LIN {X 0,Y 143.877,Z 667.344,A -85,B 0,C 180,E1 -24386.498,E2 -24386.498} C_VEL
LIN {X 0,Y 143.773,Z 666.568,A -85,B 0,C 180,E1 -24386.671,E2 -24386.671} C_VEL
LIN {X 0,Y 144.176,Z 666.526,A -85,B 0,C 180,E1 -24389.999,E2 -24389.999} C_VEL
LIN {X 0,Y 143.834,Z 666.557,A -85,B 0,C 180,E1 -24392.624,E2 -24392.624} C_VEL
LIN {X 0,Y 145.417,Z 671.126,A -85,B 0,C 180,E1 -24393.506,E2 -24393.506} C_VEL
LIN {X 0,Y 149.524,Z 680.983,A -85,B 0,C 180,E1 -24395.672,E2 -24395.672} C_VEL
LIN {X 0,Y 151.663,Z 693.614,A -85,B 0,C 180,E1 -24398.232,E2 -24398.232} C_VEL
LIN {X 0,Y 153.046,Z 704.93,A -85,B 0,C 180,E1 -24400.918,E2 -24400.918} C_VEL
LIN {X 0,Y 153.745,Z 714.71,A -85,B 0,C 180,E1 -24403.579,E2 -24403.579} C_VEL
LIN {X 0,Y 150.919,Z 725.324,A -85,B 0,C 180,E1 -24406.571,E2 -24406.571} C_VEL
LIN {X 0,Y 147.915,Z 735.227,A -85,B 0,C 180,E1 -24410.148,E2 -24410.148} C_VEL
LIN {X 0,Y 145.34,Z 743.582,A -85,B 0,C 180,E1 -24413.987,E2 -24413.987} C_VEL
LIN {X 0,Y 143.315,Z 750.513,A -85,B 0,C 180,E1 -24418.03,E2 -24418.03} C_VEL
LIN {X 0,Y 141.7,Z 756.491,A -85,B 0,C 180,E1 -24422.524,E2 -24422.524} C_VEL
LIN {X 0,Y 140.665,Z 760.98,A -85,B 0,C 180,E1 -24426.926,E2 -24426.926} C_VEL
LIN {X 0,Y 140.112,Z 764.232,A -85,B 0,C 180,E1 -24431.201,E2 -24431.201} C_VEL
LIN {X 0,Y 140.057,Z 766.475,A -85,B 0,C 180,E1 -24435.37,E2 -24435.37} C_VEL
LIN {X 0,Y 140.476,Z 767.85,A -85,B 0,C 180,E1 -24439.429,E2 -24439.429} C_VEL
LIN {X 0,Y 141.353,Z 768.412,A -85,B 0,C 180,E1 -24443.37,E2 -24443.37} C_VEL
LIN {X 0,Y 142.772,Z 768.26,A -85,B 0,C 180,E1 -24447.215,E2 -24447.215} C_VEL
LIN {X 0,Y 144.681,Z 767.428,A -85,B 0,C 180,E1 -24450.967,E2 -24450.967} C_VEL
LIN {X 0,Y 147.36,Z 765.679,A -85,B 0,C 180,E1 -24454.977,E2 -24454.977} C_VEL
LIN {X 0,Y 151.95,Z 761.946,A -85,B 0,C 180,E1 -24460.067,E2 -24460.067} C_VEL
LIN {X 0,Y 157.248,Z 757.003,A -85,B 0,C 180,E1 -24464.445,E2 -24464.445} C_VEL
LIN {X 0,Y 163.222,Z 750.532,A -85,B 0,C 180,E1 -24468.456,E2 -24468.456} C_VEL
LIN {X 0,Y 169.552,Z 742.786,A -85,B 0,C 180,E1 -24471.944,E2 -24471.944} C_VEL
LIN {X 0,Y 174.058,Z 736.389,A -85,B 0,C 180,E1 -24474.206,E2 -24474.206} C_VEL
LIN {X 0,Y 175.53,Z 732.134,A -85,B 0,C 180,E1 -24476.159,E2 -24476.159} C_VEL
LIN {X 0,Y 176.893,Z 726.441,A -85,B 0,C 180,E1 -24478.862,E2 -24478.862} C_VEL
LIN {X 0,Y 177.121,Z 724.283,A -85,B 0,C 180,E1 -24480,E2 -24480} C_VEL
LIN {X 0,Y 176.932,Z 718.916,A -85,B 0,C 180,E1 -24483.416,E2 -24483.416} C_VEL
LIN {X 0,Y 176.546,Z 715.943,A -85,B 0,C 180,E1 -24485.625,E2 -24485.625} C_VEL
LIN {X 0,Y 175.623,Z 712.219,A -85,B 0,C 180,E1 -24489.211,E2 -24489.211} C_VEL
LIN {X 0,Y 174.744,Z 708.55,A -85,B 0,C 180,E1 -24493.964,E2 -24493.964} C_VEL
LIN {X 0,Y 174.167,Z 707.771,A -85,B 0,C 180,E1 -24496.407,E2 -24496.407} C_VEL
LIN {X 0,Y 173.684,Z 707.264,A -85,B 0,C 180,E1 -24501.462,E2 -24501.462} C_VEL
LIN {X 0,Y 173.792,Z 707.475,A -85,B 0,C 180,E1 -24503.853,E2 -24503.853} C_VEL
LIN {X 0,Y 174.299,Z 708.528,A -85,B 0,C 180,E1 -24507.495,E2 -24507.495} C_VEL
LIN {X 0,Y 174.612,Z 709.116,A -85,B 0,C 180,E1 -24508.881,E2 -24508.881} C_VEL
LIN {X 0,Y 175.474,Z 712.004,A -85,B 0,C 180,E1 -24512.748,E2 -24512.748} C_VEL
LIN {X 0,Y 176.379,Z 714.975,A -85,B 0,C 180,E1 -24515.783,E2 -24515.783} C_VEL
LIN {X 0,Y 177.175,Z 718.69,A -85,B 0,C 180,E1 -24518.664,E2 -24518.664} C_VEL
LIN {X 0,Y 177.606,Z 722.793,A -85,B 0,C 180,E1 -24521.252,E2 -24521.252} C_VEL
LIN {X 0,Y 176.771,Z 726.96,A -85,B 0,C 180,E1 -24522.997,E2 -24522.997} C_VEL
LIN {X 0,Y 174.471,Z 734.554,A -85,B 0,C 180,E1 -24525.986,E2 -24525.986} C_VEL
LIN {X 0,Y 171.412,Z 742.103,A -85,B 0,C 180,E1 -24529.005,E2 -24529.005} C_VEL
LIN {X 0,Y 168.554,Z 747.562,A -85,B 0,C 180,E1 -24531.287,E2 -24531.287} C_VEL
LIN {X 0,Y 162.886,Z 754.871,A -85,B 0,C 180,E1 -24534.376,E2 -24534.376} C_VEL
LIN {X 0,Y 156.533,Z 762.037,A -85,B 0,C 180,E1 -24538.424,E2 -24538.424} C_VEL
LIN {X 0,Y 151.742,Z 767.051,A -85,B 0,C 180,E1 -24542.411,E2 -24542.411} C_VEL
LIN {X 0,Y 149.314,Z 769.45,A -85,B 0,C 180,E1 -24544.938,E2 -24544.938} C_VEL
LIN {X 0,Y 145.025,Z 773.042,A -85,B 0,C 180,E1 -24550.172,E2 -24550.172} C_VEL
LIN {X 0,Y 143.481,Z 774.261,A -85,B 0,C 180,E1 -24552.91,E2 -24552.91} C_VEL
LIN {X 0,Y 141.444,Z 775.511,A -85,B 0,C 180,E1 -24558.537,E2 -24558.537} C_VEL
LIN {X 0,Y 140.631,Z 775.285,A -85,B 0,C 180,E1 -24564.265,E2 -24564.265} C_VEL
LIN {X 0,Y 140.683,Z 774.127,A -85,B 0,C 180,E1 -24568.927,E2 -24568.927} C_VEL
LIN {X 0,Y 140.587,Z 775.783,A -85,B 0,C 180,E1 -24572.867,E2 -24572.867} C_VEL
LIN {X 0,Y 140.631,Z 776.507,A -85,B 0,C 180,E1 -24575.737,E2 -24575.737} C_VEL
LIN {X 0,Y 141.478,Z 776.775,A -85,B 0,C 180,E1 -24581.462,E2 -24581.462} C_VEL
LIN {X 0,Y 143.507,Z 775.592,A -85,B 0,C 180,E1 -24587.089,E2 -24587.089} C_VEL
LIN {X 0,Y 145.061,Z 774.441,A -85,B 0,C 180,E1 -24589.826,E2 -24589.826} C_VEL
LIN {X 0,Y 149.346,Z 770.936,A -85,B 0,C 180,E1 -24595.059,E2 -24595.059} C_VEL
LIN {X 0,Y 153.191,Z 767.268,A -85,B 0,C 180,E1 -24598.798,E2 -24598.798} C_VEL
LIN {X 0,Y 157.679,Z 762.598,A -85,B 0,C 180,E1 -24602.335,E2 -24602.335} C_VEL
LIN {X 0,Y 163.807,Z 755.698,A -85,B 0,C 180,E1 -24606.153,E2 -24606.153} C_VEL
LIN {X 0,Y 169.581,Z 748.417,A -85,B 0,C 180,E1 -24609.2,E2 -24609.2} C_VEL
LIN {X 0,Y 170.587,Z 746.519,A -85,B 0,C 180,E1 -24610.028,E2 -24610.028} C_VEL
LIN {X 0,Y 171.679,Z 743.311,A -85,B 0,C 180,E1 -24611.646,E2 -24611.646} C_VEL
LIN {X 0,Y 171.836,Z 740.481,A -85,B 0,C 180,E1 -24613.396,E2 -24613.396} C_VEL
LIN {X 0,Y 170.62,Z 732.201,A -85,B 0,C 180,E1 -24619.601,E2 -24619.601} C_VEL
LIN {X 0,Y 170.524,Z 727.368,A -85,B 0,C 180,E1 -24623.303,E2 -24623.303} C_VEL
LIN {X 0,Y 170.055,Z 723.204,A -85,B 0,C 180,E1 -24627.503,E2 -24627.503} C_VEL
LIN {X 0,Y 169.819,Z 721.041,A -85,B 0,C 180,E1 -24630.354,E2 -24630.354} C_VEL
LIN {X 0,Y 169.699,Z 719.487,A -85,B 0,C 180,E1 -24632.899,E2 -24632.899} C_VEL
LIN {X 0,Y 169.549,Z 718.56,A -85,B 0,C 180,E1 -24635.775,E2 -24635.775} C_VEL
LIN {X 0,Y 169.731,Z 718.106,A -85,B 0,C 180,E1 -24640.655,E2 -24640.655} C_VEL
LIN {X 0,Y 170.186,Z 718.227,A -85,B 0,C 180,E1 -24643.198,E2 -24643.198} C_VEL
LIN {X 0,Y 170.658,Z 720.765,A -85,B 0,C 180,E1 -24648.117,E2 -24648.117} C_VEL
LIN {X 0,Y 171.249,Z 723.52,A -85,B 0,C 180,E1 -24651.742,E2 -24651.742} C_VEL
LIN {X 0,Y 171.663,Z 726.206,A -85,B 0,C 180,E1 -24654.484,E2 -24654.484} C_VEL
LIN {X 0,Y 171.544,Z 730.318,A -85,B 0,C 180,E1 -24657.652,E2 -24657.652} C_VEL
LIN {X 0,Y 171.368,Z 732.079,A -85,B 0,C 180,E1 -24658.825,E2 -24658.825} C_VEL
LIN {X 0,Y 169.613,Z 738.213,A -85,B 0,C 180,E1 -24662.375,E2 -24662.375} C_VEL
LIN {X 0,Y 168.953,Z 739.907,A -85,B 0,C 180,E1 -24663.296,E2 -24663.296} C_VEL
LIN {X 0,Y 167.061,Z 742.729,A -85,B 0,C 180,E1 -24664.453,E2 -24664.453} C_VEL
LIN {X 0,Y 160.74,Z 750.003,A -85,B 0,C 180,E1 -24667.537,E2 -24667.537} C_VEL
LIN {X 0,Y 154.586,Z 756.204,A -85,B 0,C 180,E1 -24671.08,E2 -24671.08} C_VEL
LIN {X 0,Y 149.083,Z 761.155,A -85,B 0,C 180,E1 -24675.027,E2 -24675.027} C_VEL
LIN {X 0,Y 143.481,Z 765.467,A -85,B 0,C 180,E1 -24680.052,E2 -24680.052} C_VEL
LIN {X 0,Y 139.494,Z 767.958,A -85,B 0,C 180,E1 -24684.921,E2 -24684.921} C_VEL
LIN {X 0,Y 135.948,Z 769.379,A -85,B 0,C 180,E1 -24691.129,E2 -24691.129} C_VEL
LIN {X 0,Y 134.47,Z 769.341,A -85,B 0,C 180,E1 -24695.094,E2 -24695.094} C_VEL
LIN {X 0,Y 133.553,Z 768.642,A -85,B 0,C 180,E1 -24699.16,E2 -24699.16} C_VEL
LIN {X 0,Y 133.064,Z 767.199,A -85,B 0,C 180,E1 -24703.363,E2 -24703.363} C_VEL
LIN {X 0,Y 133.302,Z 763.826,A -85,B 0,C 180,E1 -24709.258,E2 -24709.258} C_VEL
LIN {X 0,Y 133.964,Z 760.423,A -85,B 0,C 180,E1 -24713.451,E2 -24713.451} C_VEL
LIN {X 0,Y 135.282,Z 754.735,A -85,B 0,C 180,E1 -24718.699,E2 -24718.699} C_VEL
LIN {X 0,Y 137.191,Z 748.084,A -85,B 0,C 180,E1 -24723.369,E2 -24723.369} C_VEL
LIN {X 0,Y 139.824,Z 739.765,A -85,B 0,C 180,E1 -24727.852,E2 -24727.852} C_VEL
LIN {X 0,Y 142.721,Z 730.618,A -85,B 0,C 180,E1 -24731.703,E2 -24731.703} C_VEL
LIN {X 0,Y 145.849,Z 720.501,A -85,B 0,C 180,E1 -24735.031,E2 -24735.031} C_VEL
LIN {X 0,Y 146.973,Z 716.437,A -85,B 0,C 180,E1 -24736.166,E2 -24736.166} C_VEL
LIN {X 0,Y 146.105,Z 705.581,A -85,B 0,C 180,E1 -24739.328,E2 -24739.328} C_VEL
LIN {X 0,Y 144.521,Z 693.495,A -85,B 0,C 180,E1 -24742.384,E2 -24742.384} C_VEL
LIN {X 0,Y 142.148,Z 681.493,A -85,B 0,C 180,E1 -24745.035,E2 -24745.035} C_VEL
LIN {X 0,Y 140.918,Z 677.424,A -85,B 0,C 180,E1 -24745.918,E2 -24745.918} C_VEL
LIN {X 0,Y 136.942,Z 668.016,A -85,B 0,C 180,E1 -24748.069,E2 -24748.069} C_VEL
LIN {X 0,Y 136.854,Z 667.433,A -85,B 0,C 180,E1 -24748.159,E2 -24748.159} C_VEL
LIN {X 0,Y 137.013,Z 667.415,A -85,B 0,C 180,E1 -24750.734,E2 -24750.734} C_VEL
LIN {X 0,Y 136.955,Z 667.42,A -85,B 0,C 180,E1 -24751.101,E2 -24751.101} C_VEL
LIN {X 0,Y 137.916,Z 670.303,A -85,B 0,C 180,E1 -24751.687,E2 -24751.687} C_VEL
LIN {X 0,Y 142.947,Z 682.693,A -85,B 0,C 180,E1 -24754.58,E2 -24754.58} C_VEL
LIN {X 0,Y 144.87,Z 693.242,A -85,B 0,C 180,E1 -24756.879,E2 -24756.879} C_VEL
LIN {X 0,Y 146.171,Z 704.573,A -85,B 0,C 180,E1 -24759.687,E2 -24759.687} C_VEL
LIN {X 0,Y 146.911,Z 715.361,A -85,B 0,C 180,E1 -24762.781,E2 -24762.781} C_VEL
LIN {X 0,Y 144.859,Z 723.128,A -85,B 0,C 180,E1 -24765.026,E2 -24765.026} C_VEL
LIN {X 0,Y 141.727,Z 733.249,A -85,B 0,C 180,E1 -24768.608,E2 -24768.608} C_VEL
LIN {X 0,Y 139.064,Z 741.396,A -85,B 0,C 180,E1 -24772.272,E2 -24772.272} C_VEL
LIN {X 0,Y 136.701,Z 749.132,A -85,B 0,C 180,E1 -24776.733,E2 -24776.733} C_VEL
LIN {X 0,Y 134.89,Z 755.433,A -85,B 0,C 180,E1 -24781.399,E2 -24781.399} C_VEL
LIN {X 0,Y 133.651,Z 760.641,A -85,B 0,C 180,E1 -24786.507,E2 -24786.507} C_VEL
LIN {X 0,Y 132.946,Z 764.78,A -85,B 0,C 180,E1 -24792.261,E2 -24792.261} C_VEL
LIN {X 0,Y 133.115,Z 767.283,A -85,B 0,C 180,E1 -24797.657,E2 -24797.657} C_VEL
LIN {X 0,Y 133.863,Z 768.35,A -85,B 0,C 180,E1 -24801.952,E2 -24801.952} C_VEL
LIN {X 0,Y 135.187,Z 768.647,A -85,B 0,C 180,E1 -24806.281,E2 -24806.281} C_VEL
LIN {X 0,Y 137.18,Z 768.142,A -85,B 0,C 180,E1 -24810.565,E2 -24810.565} C_VEL
LIN {X 0,Y 141.189,Z 765.96,A -85,B 0,C 180,E1 -24816.533,E2 -24816.533} C_VEL
LIN {X 0,Y 145.889,Z 762.517,A -85,B 0,C 180,E1 -24821.495,E2 -24821.495} C_VEL
LIN {X 0,Y 151.913,Z 757.345,A -85,B 0,C 180,E1 -24826.289,E2 -24826.289} C_VEL
LIN {X 0,Y 157.186,Z 752.125,A -85,B 0,C 180,E1 -24829.697,E2 -24829.697} C_VEL
LIN {X 0,Y 164.111,Z 744.275,A -85,B 0,C 180,E1 -24833.434,E2 -24833.434} C_VEL
LIN {X 0,Y 167.966,Z 739.5,A -85,B 0,C 180,E1 -24835.2,E2 -24835.2} C_VEL
LIN {X 0,Y 169.073,Z 737.548,A -85,B 0,C 180,E1 -24836.032,E2 -24836.032} C_VEL
LIN {X 0,Y 171.356,Z 730.897,A -85,B 0,C 180,E1 -24839.412,E2 -24839.412} C_VEL
LIN {X 0,Y 171.934,Z 727.872,A -85,B 0,C 180,E1 -24841.171,E2 -24841.171} C_VEL
LIN {X 0,Y 172.047,Z 722.847,A -85,B 0,C 180,E1 -24844.686,E2 -24844.686} C_VEL
LIN {X 0,Y 171.772,Z 720.188,A -85,B 0,C 180,E1 -24847.05,E2 -24847.05} C_VEL
LIN {X 0,Y 171.276,Z 717.469,A -85,B 0,C 180,E1 -24850.011,E2 -24850.011} C_VEL
LIN {X 0,Y 170.821,Z 714.422,A -85,B 0,C 180,E1 -24854.291,E2 -24854.291} C_VEL
LIN {X 0,Y 170.129,Z 713.525,A -85,B 0,C 180,E1 -24858.176,E2 -24858.176} C_VEL
LIN {X 0,Y 169.983,Z 713.327,A -85,B 0,C 180,E1 -24861.846,E2 -24861.846} C_VEL
LIN {X 0,Y 170.123,Z 713.691,A -85,B 0,C 180,E1 -24864.657,E2 -24864.657} C_VEL
LIN {X 0,Y 170.445,Z 714.362,A -85,B 0,C 180,E1 -24866.973,E2 -24866.973} C_VEL
LIN {X 0,Y 170.991,Z 716.137,A -85,B 0,C 180,E1 -24870.333,E2 -24870.333} C_VEL
LIN {X 0,Y 171.931,Z 719.941,A -85,B 0,C 180,E1 -24874.909,E2 -24874.909} C_VEL
LIN {X 0,Y 172.494,Z 724.271,A -85,B 0,C 180,E1 -24878.489,E2 -24878.489} C_VEL
LIN {X 0,Y 172.469,Z 727.696,A -85,B 0,C 180,E1 -24880.692,E2 -24880.692} C_VEL
LIN {X 0,Y 170.079,Z 734.784,A -85,B 0,C 180,E1 -24883.688,E2 -24883.688} C_VEL
LIN {X 0,Y 167.014,Z 741.744,A -85,B 0,C 180,E1 -24886.648,E2 -24886.648} C_VEL
LIN {X 0,Y 163.986,Z 747.466,A -85,B 0,C 180,E1 -24889.19,E2 -24889.19} C_VEL
LIN {X 0,Y 158.209,Z 754.666,A -85,B 0,C 180,E1 -24892.354,E2 -24892.354} C_VEL
LIN {X 0,Y 151.712,Z 761.502,A -85,B 0,C 180,E1 -24896.229,E2 -24896.229} C_VEL
LIN {X 0,Y 146.898,Z 766.135,A -85,B 0,C 180,E1 -24899.846,E2 -24899.846} C_VEL
LIN {X 0,Y 142.9,Z 769.737,A -85,B 0,C 180,E1 -24903.73,E2 -24903.73} C_VEL
LIN {X 0,Y 138.364,Z 773.15,A -85,B 0,C 180,E1 -24909.174,E2 -24909.174} C_VEL
LIN {X 0,Y 135.422,Z 774.977,A -85,B 0,C 180,E1 -24914.962,E2 -24914.962} C_VEL
LIN {X 0,Y 133.868,Z 775.348,A -85,B 0,C 180,E1 -24920.94,E2 -24920.94} C_VEL
LIN {X 0,Y 133.555,Z 774.956,A -85,B 0,C 180,E1 -24923.96,E2 -24923.96} C_VEL
LIN {X 0,Y 133.602,Z 773.586,A -85,B 0,C 180,E1 -24928.872,E2 -24928.872} C_VEL
LIN {X 0,Y 133.512,Z 775.326,A -85,B 0,C 180,E1 -24933.019,E2 -24933.019} C_VEL
LIN {X 0,Y 133.878,Z 776.564,A -85,B 0,C 180,E1 -24939.062,E2 -24939.062} C_VEL
LIN {X 0,Y 135.436,Z 776.253,A -85,B 0,C 180,E1 -24945.039,E2 -24945.039} C_VEL
LIN {X 0,Y 138.399,Z 774.501,A -85,B 0,C 180,E1 -24950.823,E2 -24950.823} C_VEL
LIN {X 0,Y 140.504,Z 773.076,A -85,B 0,C 180,E1 -24953.589,E2 -24953.589} C_VEL
LIN {X 0,Y 145.597,Z 768.98,A -85,B 0,C 180,E1 -24958.863,E2 -24958.863} C_VEL
LIN {X 0,Y 149.74,Z 765.144,A -85,B 0,C 180,E1 -24962.347,E2 -24962.347} C_VEL
LIN {X 0,Y 155.32,Z 759.646,A -85,B 0,C 180,E1 -24966.033,E2 -24966.033} C_VEL
LIN {X 0,Y 162.173,Z 752.08,A -85,B 0,C 180,E1 -24969.734,E2 -24969.734} C_VEL
LIN {X 0,Y 164.164,Z 749.58,A -85,B 0,C 180,E1 -24970.759,E2 -24970.759} C_VEL
LIN {X 0,Y 166.941,Z 744.35,A -85,B 0,C 180,E1 -24973.256,E2 -24973.256} C_VEL
LIN {X 0,Y 169.559,Z 737.815,A -85,B 0,C 180,E1 -24976.388,E2 -24976.388} C_VEL
LIN {X 0,Y 170.382,Z 734.81,A -85,B 0,C 180,E1 -24977.943,E2 -24977.943} C_VEL
LIN {X 0,Y 170.62,Z 732.201,A -85,B 0,C 180,E1 -24979.601,E2 -24979.601} C_VEL
LIN {X 0,Y 170.448,Z 730.742,A -85,B 0,C 180,E1 -24980.824,E2 -24980.824} C_VEL
LIN {X 0,Y 169.873,Z 729.73,A -85,B 0,C 180,E1 -24982.09,E2 -24982.09} C_VEL
LIN {X 0,Y 168.084,Z 728.621,A -85,B 0,C 180,E1 -24984.691,E2 -24984.691} C_VEL
LIN {X 0,Y 165.588,Z 727.537,A -85,B 0,C 180,E1 -24988.78,E2 -24988.78} C_VEL
LIN {X 0,Y 165.312,Z 726.849,A -85,B 0,C 180,E1 -24990.162,E2 -24990.162} C_VEL
LIN {X 0,Y 165.344,Z 725.034,A -85,B 0,C 180,E1 -24993.205,E2 -24993.205} C_VEL
LIN {X 0,Y 165.222,Z 723.985,A -85,B 0,C 180,E1 -24997.491,E2 -24997.491} C_VEL
LIN {X 0,Y 165.784,Z 723.848,A -85,B 0,C 180,E1 -25002.738,E2 -25002.738} C_VEL
LIN {X 0,Y 166.076,Z 726.08,A -85,B 0,C 180,E1 -25007.784,E2 -25007.784} C_VEL
LIN {X 0,Y 166.353,Z 727.748,A -85,B 0,C 180,E1 -25010.271,E2 -25010.271} C_VEL
LIN {X 0,Y 166.608,Z 730.901,A -85,B 0,C 180,E1 -25013.947,E2 -25013.947} C_VEL
LIN {X 0,Y 166.03,Z 735.341,A -85,B 0,C 180,E1 -25017.574,E2 -25017.574} C_VEL
LIN {X 0,Y 164.813,Z 739.113,A -85,B 0,C 180,E1 -25020,E2 -25020} C_VEL
LIN {X 0,Y 163.548,Z 742.116,A -85,B 0,C 180,E1 -25021.847,E2 -25021.847} C_VEL
LIN {X 0,Y 162.481,Z 743.669,A -85,B 0,C 180,E1 -25022.585,E2 -25022.585} C_VEL
LIN {X 0,Y 155.436,Z 751.174,A -85,B 0,C 180,E1 -25025.881,E2 -25025.881} C_VEL
LIN {X 0,Y 149.498,Z 756.743,A -85,B 0,C 180,E1 -25029.165,E2 -25029.165} C_VEL
LIN {X 0,Y 144.136,Z 761.223,A -85,B 0,C 180,E1 -25032.786,E2 -25032.786} C_VEL
LIN {X 0,Y 138.177,Z 765.486,A -85,B 0,C 180,E1 -25037.769,E2 -25037.769} C_VEL
LIN {X 0,Y 134.752,Z 767.488,A -85,B 0,C 180,E1 -25041.413,E2 -25041.413} C_VEL
LIN {X 0,Y 131.938,Z 768.853,A -85,B 0,C 180,E1 -25045.223,E2 -25045.223} C_VEL
LIN {X 0,Y 129.404,Z 769.619,A -85,B 0,C 180,E1 -25049.659,E2 -25049.659} C_VEL
LIN {X 0,Y 127.561,Z 769.54,A -85,B 0,C 180,E1 -25054.265,E2 -25054.265} C_VEL
LIN {X 0,Y 126.474,Z 768.651,A -85,B 0,C 180,E1 -25058.924,E2 -25058.924} C_VEL
LIN {X 0,Y 125.954,Z 766.998,A -85,B 0,C 180,E1 -25063.498,E2 -25063.498} C_VEL
LIN {X 0,Y 126.262,Z 763.438,A -85,B 0,C 180,E1 -25069.684,E2 -25069.684} C_VEL
LIN {X 0,Y 127.015,Z 759.696,A -85,B 0,C 180,E1 -25074.261,E2 -25074.261} C_VEL
LIN {X 0,Y 128.421,Z 753.981,A -85,B 0,C 180,E1 -25079.586,E2 -25079.586} C_VEL
LIN {X 0,Y 130.529,Z 747.046,A -85,B 0,C 180,E1 -25084.484,E2 -25084.484} C_VEL
LIN {X 0,Y 133.116,Z 739.143,A -85,B 0,C 180,E1 -25088.841,E2 -25088.841} C_VEL
LIN {X 0,Y 136.06,Z 730.262,A -85,B 0,C 180,E1 -25092.698,E2 -25092.698} C_VEL
LIN {X 0,Y 139.324,Z 720.091,A -85,B 0,C 180,E1 -25096.135,E2 -25096.135} C_VEL
LIN {X 0,Y 140.144,Z 717.281,A -85,B 0,C 180,E1 -25096.957,E2 -25096.957} C_VEL
LIN {X 0,Y 139.415,Z 706.773,A -85,B 0,C 180,E1 -25100.203,E2 -25100.203} C_VEL
LIN {X 0,Y 137.9,Z 694.621,A -85,B 0,C 180,E1 -25103.461,E2 -25103.461} C_VEL
LIN {X 0,Y 135.55,Z 682.141,A -85,B 0,C 180,E1 -25106.424,E2 -25106.424} C_VEL
LIN {X 0,Y 130.357,Z 669.741,A -85,B 0,C 180,E1 -25109.68,E2 -25109.68} C_VEL
LIN {X 0,Y 133.526,Z 677.164,A -85,B 0,C 180,E1 -25111.525,E2 -25111.525} C_VEL
LIN {X 0,Y 137.162,Z 686.775,A -85,B 0,C 180,E1 -25114.037,E2 -25114.037} C_VEL
LIN {X 0,Y 138.804,Z 698.646,A -85,B 0,C 180,E1 -25116.878,E2 -25116.878} C_VEL
LIN {X 0,Y 139.787,Z 709.084,A -85,B 0,C 180,E1 -25119.768,E2 -25119.768} C_VEL
LIN {X 0,Y 140.129,Z 716.082,A -85,B 0,C 180,E1 -25121.939,E2 -25121.939} C_VEL
LIN {X 0,Y 137.462,Z 725.362,A -85,B 0,C 180,E1 -25124.81,E2 -25124.81} C_VEL
LIN {X 0,Y 134.526,Z 734.345,A -85,B 0,C 180,E1 -25128.266,E2 -25128.266} C_VEL
LIN {X 0,Y 131.413,Z 743.733,A -85,B 0,C 180,E1 -25132.932,E2 -25132.932} C_VEL
LIN {X 0,Y 129.237,Z 750.581,A -85,B 0,C 180,E1 -25137.307,E2 -25137.307} C_VEL
LIN {X 0,Y 127.4,Z 756.884,A -85,B 0,C 180,E1 -25142.536,E2 -25142.536} C_VEL
LIN {X 0,Y 126.292,Z 761.608,A -85,B 0,C 180,E1 -25147.742,E2 -25147.742} C_VEL
LIN {X 0,Y 125.821,Z 765.318,A -85,B 0,C 180,E1 -25153.436,E2 -25153.436} C_VEL
LIN {X 0,Y 126.043,Z 767.289,A -85,B 0,C 180,E1 -25158.002,E2 -25158.002} C_VEL
LIN {X 0,Y 126.84,Z 768.452,A -85,B 0,C 180,E1 -25162.447,E2 -25162.447} C_VEL
LIN {X 0,Y 128.172,Z 768.891,A -85,B 0,C 180,E1 -25166.748,E2 -25166.748} C_VEL
LIN {X 0,Y 130.105,Z 768.588,A -85,B 0,C 180,E1 -25170.911,E2 -25170.911} C_VEL
LIN {X 0,Y 132.548,Z 767.618,A -85,B 0,C 180,E1 -25174.901,E2 -25174.901} C_VEL
LIN {X 0,Y 137.358,Z 764.891,A -85,B 0,C 180,E1 -25180.615,E2 -25180.615} C_VEL
LIN {X 0,Y 141.507,Z 761.966,A -85,B 0,C 180,E1 -25184.359,E2 -25184.359} C_VEL
LIN {X 0,Y 146.147,Z 758.213,A -85,B 0,C 180,E1 -25187.853,E2 -25187.853} C_VEL
LIN {X 0,Y 153.053,Z 751.892,A -85,B 0,C 180,E1 -25192.082,E2 -25192.082} C_VEL
LIN {X 0,Y 159.595,Z 744.95,A -85,B 0,C 180,E1 -25195.378,E2 -25195.378} C_VEL
LIN {X 0,Y 162.682,Z 741.371,A -85,B 0,C 180,E1 -25196.729,E2 -25196.729} C_VEL
LIN {X 0,Y 164.307,Z 738.485,A -85,B 0,C 180,E1 -25198.162,E2 -25198.162} C_VEL
LIN {X 0,Y 166.08,Z 734.091,A -85,B 0,C 180,E1 -25200.606,E2 -25200.606} C_VEL
LIN {X 0,Y 166.704,Z 731.342,A -85,B 0,C 180,E1 -25202.416,E2 -25202.416} C_VEL
LIN {X 0,Y 167.111,Z 726.762,A -85,B 0,C 180,E1 -25206.035,E2 -25206.035} C_VEL
LIN {X 0,Y 166.864,Z 723.391,A -85,B 0,C 180,E1 -25209.699,E2 -25209.699} C_VEL
LIN {X 0,Y 166.621,Z 720.076,A -85,B 0,C 180,E1 -25214.66,E2 -25214.66} C_VEL
LIN {X 0,Y 165.949,Z 719.221,A -85,B 0,C 180,E1 -25219.804,E2 -25219.804} C_VEL
LIN {X 0,Y 165.967,Z 719.235,A -85,B 0,C 180,E1 -25222.402,E2 -25222.402} C_VEL
LIN {X 0,Y 166.122,Z 719.636,A -85,B 0,C 180,E1 -25225.028,E2 -25225.028} C_VEL
LIN {X 0,Y 166.418,Z 720.531,A -85,B 0,C 180,E1 -25227.68,E2 -25227.68} C_VEL
LIN {X 0,Y 166.775,Z 721.998,A -85,B 0,C 180,E1 -25230.377,E2 -25230.377} C_VEL
LIN {X 0,Y 167.145,Z 723.993,A -85,B 0,C 180,E1 -25233.135,E2 -25233.135} C_VEL
LIN {X 0,Y 167.497,Z 726.775,A -85,B 0,C 180,E1 -25235.975,E2 -25235.975} C_VEL
LIN {X 0,Y 167.524,Z 730.545,A -85,B 0,C 180,E1 -25238.997,E2 -25238.997} C_VEL
LIN {X 0,Y 166.55,Z 733.604,A -85,B 0,C 180,E1 -25240.577,E2 -25240.577} C_VEL
LIN {X 0,Y 163.776,Z 739.805,A -85,B 0,C 180,E1 -25243.361,E2 -25243.361} C_VEL
LIN {X 0,Y 159.501,Z 747.442,A -85,B 0,C 180,E1 -25246.926,E2 -25246.926} C_VEL
LIN {X 0,Y 156.8,Z 751.083,A -85,B 0,C 180,E1 -25248.617,E2 -25248.617} C_VEL
LIN {X 0,Y 149.685,Z 758.609,A -85,B 0,C 180,E1 -25252.385,E2 -25252.385} C_VEL
LIN {X 0,Y 143.169,Z 764.611,A -85,B 0,C 180,E1 -25256.565,E2 -25256.565} C_VEL
LIN {X 0,Y 137.914,Z 768.99,A -85,B 0,C 180,E1 -25261.047,E2 -25261.047} C_VEL
LIN {X 0,Y 133.989,Z 771.836,A -85,B 0,C 180,E1 -25265.191,E2 -25265.191} C_VEL
LIN {X 0,Y 129.911,Z 774.23,A -85,B 0,C 180,E1 -25271.061,E2 -25271.061} C_VEL
LIN {X 0,Y 127.509,Z 775.175,A -85,B 0,C 180,E1 -25277.265,E2 -25277.265} C_VEL
LIN {X 0,Y 126.503,Z 774.577,A -85,B 0,C 180,E1 -25283.622,E2 -25283.622} C_VEL
LIN {X 0,Y 126.532,Z 772.979,A -85,B 0,C 180,E1 -25288.809,E2 -25288.809} C_VEL
LIN {X 0,Y 126.438,Z 774.863,A -85,B 0,C 180,E1 -25293.188,E2 -25293.188} C_VEL
LIN {X 0,Y 126.866,Z 776.248,A -85,B 0,C 180,E1 -25299.568,E2 -25299.568} C_VEL
LIN {X 0,Y 128.574,Z 776.15,A -85,B 0,C 180,E1 -25305.862,E2 -25305.862} C_VEL
LIN {X 0,Y 131.788,Z 774.555,A -85,B 0,C 180,E1 -25311.92,E2 -25311.92} C_VEL
LIN {X 0,Y 136.601,Z 771.496,A -85,B 0,C 180,E1 -25317.585,E2 -25317.585} C_VEL
LIN {X 0,Y 140.916,Z 768.16,A -85,B 0,C 180,E1 -25321.58,E2 -25321.58} C_VEL
LIN {X 0,Y 145.934,Z 763.87,A -85,B 0,C 180,E1 -25325.305,E2 -25325.305} C_VEL
LIN {X 0,Y 152.682,Z 757.526,A -85,B 0,C 180,E1 -25329.267,E2 -25329.267} C_VEL
LIN {X 0,Y 158.879,Z 750.784,A -85,B 0,C 180,E1 -25332.423,E2 -25332.423} C_VEL
LIN {X 0,Y 162.439,Z 744.573,A -85,B 0,C 180,E1 -25335.621,E2 -25335.621} C_VEL
LIN {X 0,Y 164.513,Z 739.834,A -85,B 0,C 180,E1 -25338.112,E2 -25338.112} C_VEL
LIN {X 0,Y 165.254,Z 736.923,A -85,B 0,C 180,E1 -25339.954,E2 -25339.954} C_VEL
LIN {X 0,Y 165.52,Z 733.712,A -85,B 0,C 180,E1 -25342.46,E2 -25342.46} C_VEL
LIN {X 0,Y 165.476,Z 729.624,A -85,B 0,C 180,E1 -25346.487,E2 -25346.487} C_VEL
LIN {X 0,Y 165.312,Z 726.849,A -85,B 0,C 180,E1 -25350.162,E2 -25350.162} C_VEL
LIN {X 0,Y 164.797,Z 726.267,A -85,B 0,C 180,E1 -25352.188,E2 -25352.188} C_VEL
LIN {X 0,Y 163.719,Z 726.659,A -85,B 0,C 180,E1 -25354.223,E2 -25354.223} C_VEL
LIN {X 0,Y 160.99,Z 729.081,A -85,B 0,C 180,E1 -25359.769,E2 -25359.769} C_VEL
LIN {X 0,Y 160.958,Z 729.275,A -85,B 0,C 180,E1 -25361.202,E2 -25361.202} C_VEL
LIN {X 0,Y 161.125,Z 729.272,A -85,B 0,C 180,E1 -25362.222,E2 -25362.222} C_VEL
LIN {X 0,Y 161.264,Z 731.19,A -85,B 0,C 180,E1 -25367.414,E2 -25367.414} C_VEL
LIN {X 0,Y 161.375,Z 732.762,A -85,B 0,C 180,E1 -25369.968,E2 -25369.968} C_VEL
LIN {X 0,Y 161.296,Z 735.788,A -85,B 0,C 180,E1 -25373.746,E2 -25373.746} C_VEL
LIN {X 0,Y 160.697,Z 738.558,A -85,B 0,C 180,E1 -25376.239,E2 -25376.239} C_VEL
LIN {X 0,Y 159.346,Z 741.95,A -85,B 0,C 180,E1 -25378.736,E2 -25378.736} C_VEL
LIN {X 0,Y 158.447,Z 743.831,A -85,B 0,C 180,E1 -25380,E2 -25380} C_VEL
LIN {X 0,Y 157.19,Z 745.639,A -85,B 0,C 180,E1 -25381.005,E2 -25381.005} C_VEL
LIN {X 0,Y 150.788,Z 751.967,A -85,B 0,C 180,E1 -25383.876,E2 -25383.876} C_VEL
LIN {X 0,Y 143.529,Z 758.188,A -85,B 0,C 180,E1 -25387.739,E2 -25387.739} C_VEL
LIN {X 0,Y 136.709,Z 763.211,A -85,B 0,C 180,E1 -25392.372,E2 -25392.372} C_VEL
LIN {X 0,Y 131.885,Z 766.206,A -85,B 0,C 180,E1 -25396.421,E2 -25396.421} C_VEL
LIN {X 0,Y 127.784,Z 768.303,A -85,B 0,C 180,E1 -25400.771,E2 -25400.771} C_VEL
LIN {X 0,Y 123.447,Z 769.754,A -85,B 0,C 180,E1 -25407.094,E2 -25407.094} C_VEL
LIN {X 0,Y 121.427,Z 769.875,A -85,B 0,C 180,E1 -25411.393,E2 -25411.393} C_VEL
LIN {X 0,Y 119.971,Z 769.33,A -85,B 0,C 180,E1 -25415.86,E2 -25415.86} C_VEL
LIN {X 0,Y 119.116,Z 768.045,A -85,B 0,C 180,E1 -25420.468,E2 -25420.468} C_VEL
LIN {X 0,Y 118.833,Z 766,A -85,B 0,C 180,E1 -25425.211,E2 -25425.211} C_VEL
LIN {X 0,Y 119.192,Z 763.094,A -85,B 0,C 180,E1 -25430.044,E2 -25430.044} C_VEL
LIN {X 0,Y 120.041,Z 759.05,A -85,B 0,C 180,E1 -25435.051,E2 -25435.051} C_VEL
LIN {X 0,Y 121.463,Z 753.575,A -85,B 0,C 180,E1 -25440.218,E2 -25440.218} C_VEL
LIN {X 0,Y 123.718,Z 746.522,A -85,B 0,C 180,E1 -25445.356,E2 -25445.356} C_VEL
LIN {X 0,Y 126.803,Z 737.463,A -85,B 0,C 180,E1 -25450.429,E2 -25450.429} C_VEL
LIN {X 0,Y 129.904,Z 728.441,A -85,B 0,C 180,E1 -25454.304,E2 -25454.304} C_VEL
LIN {X 0,Y 133.315,Z 717.96,A -85,B 0,C 180,E1 -25457.825,E2 -25457.825} C_VEL
LIN {X 0,Y 132.809,Z 708.787,A -85,B 0,C 180,E1 -25460.864,E2 -25460.864} C_VEL
LIN {X 0,Y 131.728,Z 698.59,A -85,B 0,C 180,E1 -25463.873,E2 -25463.873} C_VEL
LIN {X 0,Y 129.877,Z 687.118,A -85,B 0,C 180,E1 -25466.897,E2 -25466.897} C_VEL
LIN {X 0,Y 129.073,Z 684.164,A -85,B 0,C 180,E1 -25467.658,E2 -25467.658} C_VEL
LIN {X 0,Y 126.313,Z 677.321,A -85,B 0,C 180,E1 -25469.6,E2 -25469.6} C_VEL
LIN {X 0,Y 130.916,Z 689.346,A -85,B 0,C 180,E1 -25473.076,E2 -25473.076} C_VEL
LIN {X 0,Y 132.323,Z 700.868,A -85,B 0,C 180,E1 -25476.096,E2 -25476.096} C_VEL
LIN {X 0,Y 133.172,Z 712.129,A -85,B 0,C 180,E1 -25479.491,E2 -25479.491} C_VEL
LIN {X 0,Y 133.341,Z 716.673,A -85,B 0,C 180,E1 -25481.013,E2 -25481.013} C_VEL
LIN {X 0,Y 130.456,Z 726.233,A -85,B 0,C 180,E1 -25484.138,E2 -25484.138} C_VEL
LIN {X 0,Y 127.514,Z 734.811,A -85,B 0,C 180,E1 -25487.645,E2 -25487.645} C_VEL
LIN {X 0,Y 124.382,Z 743.921,A -85,B 0,C 180,E1 -25492.419,E2 -25492.419} C_VEL
LIN {X 0,Y 121.955,Z 751.311,A -85,B 0,C 180,E1 -25497.451,E2 -25497.451} C_VEL
LIN {X 0,Y 120.125,Z 757.683,A -85,B 0,C 180,E1 -25503.199,E2 -25503.199} C_VEL
LIN {X 0,Y 119.153,Z 761.648,A -85,B 0,C 180,E1 -25507.896,E2 -25507.896} C_VEL
LIN {X 0,Y 118.746,Z 764.706,A -85,B 0,C 180,E1 -25512.638,E2 -25512.638} C_VEL
LIN {X 0,Y 119.128,Z 767.674,A -85,B 0,C 180,E1 -25519.537,E2 -25519.537} C_VEL
LIN {X 0,Y 120.326,Z 768.848,A -85,B 0,C 180,E1 -25524.854,E2 -25524.854} C_VEL
LIN {X 0,Y 122.176,Z 769.075,A -85,B 0,C 180,E1 -25529.635,E2 -25529.635} C_VEL
LIN {X 0,Y 124.775,Z 768.507,A -85,B 0,C 180,E1 -25534.313,E2 -25534.313} C_VEL
LIN {X 0,Y 128.118,Z 767.118,A -85,B 0,C 180,E1 -25538.83,E2 -25538.83} C_VEL
LIN {X 0,Y 132.223,Z 764.879,A -85,B 0,C 180,E1 -25543.081,E2 -25543.081} C_VEL
LIN {X 0,Y 138.738,Z 760.479,A -85,B 0,C 180,E1 -25548.309,E2 -25548.309} C_VEL
LIN {X 0,Y 145.002,Z 755.479,A -85,B 0,C 180,E1 -25552.285,E2 -25552.285} C_VEL
LIN {X 0,Y 152.162,Z 748.828,A -85,B 0,C 180,E1 -25556.028,E2 -25556.028} C_VEL
LIN {X 0,Y 158.072,Z 742.516,A -85,B 0,C 180,E1 -25558.726,E2 -25558.726} C_VEL
LIN {X 0,Y 160.358,Z 738.192,A -85,B 0,C 180,E1 -25561.256,E2 -25561.256} C_VEL
LIN {X 0,Y 161.051,Z 736.348,A -85,B 0,C 180,E1 -25562.501,E2 -25562.501} C_VEL
LIN {X 0,Y 161.762,Z 733.257,A -85,B 0,C 180,E1 -25564.985,E2 -25564.985} C_VEL
LIN {X 0,Y 162.062,Z 730.628,A -85,B 0,C 180,E1 -25567.475,E2 -25567.475} C_VEL
LIN {X 0,Y 162.087,Z 728.618,A -85,B 0,C 180,E1 -25569.988,E2 -25569.988} C_VEL
LIN {X 0,Y 162.107,Z 725.511,A -85,B 0,C 180,E1 -25575.077,E2 -25575.077} C_VEL
LIN {X 0,Y 161.607,Z 724.818,A -85,B 0,C 180,E1 -25580.359,E2 -25580.359} C_VEL
LIN {X 0,Y 161.695,Z 725.122,A -85,B 0,C 180,E1 -25584.114,E2 -25584.114} C_VEL
LIN {X 0,Y 161.833,Z 725.483,A -85,B 0,C 180,E1 -25585.739,E2 -25585.739} C_VEL
LIN {X 0,Y 162.182,Z 727.278,A -85,B 0,C 180,E1 -25589.928,E2 -25589.928} C_VEL
LIN {X 0,Y 162.428,Z 729.161,A -85,B 0,C 180,E1 -25592.74,E2 -25592.74} C_VEL
LIN {X 0,Y 162.53,Z 731.898,A -85,B 0,C 180,E1 -25595.714,E2 -25595.714} C_VEL
LIN {X 0,Y 162.41,Z 733.652,A -85,B 0,C 180,E1 -25597.288,E2 -25597.288} C_VEL
LIN {X 0,Y 161.988,Z 735.613,A -85,B 0,C 180,E1 -25598.655,E2 -25598.655} C_VEL
LIN {X 0,Y 158.981,Z 741.459,A -85,B 0,C 180,E1 -25601.537,E2 -25601.537} C_VEL
LIN {X 0,Y 154.397,Z 748.701,A -85,B 0,C 180,E1 -25605.128,E2 -25605.128} C_VEL
LIN {X 0,Y 152.677,Z 751.043,A -85,B 0,C 180,E1 -25606.334,E2 -25606.334} C_VEL
LIN {X 0,Y 146.263,Z 757.513,A -85,B 0,C 180,E1 -25609.56,E2 -25609.56} C_VEL
LIN {X 0,Y 140.214,Z 762.815,A -85,B 0,C 180,E1 -25613.026,E2 -25613.026} C_VEL
LIN {X 0,Y 135.429,Z 766.625,A -85,B 0,C 180,E1 -25616.348,E2 -25616.348} C_VEL
LIN {X 0,Y 130.289,Z 770.323,A -85,B 0,C 180,E1 -25620.958,E2 -25620.958} C_VEL
LIN {X 0,Y 125.175,Z 773.284,A -85,B 0,C 180,E1 -25626.859,E2 -25626.859} C_VEL
LIN {X 0,Y 123.19,Z 774.221,A -85,B 0,C 180,E1 -25629.984,E2 -25629.984} C_VEL
LIN {X 0,Y 120.571,Z 774.946,A -85,B 0,C 180,E1 -25636.518,E2 -25636.518} C_VEL
LIN {X 0,Y 119.442,Z 774.198,A -85,B 0,C 180,E1 -25643.243,E2 -25643.243} C_VEL
LIN {X 0,Y 119.459,Z 772.51,A -85,B 0,C 180,E1 -25649.012,E2 -25649.012} C_VEL
LIN {X 0,Y 119.354,Z 774.388,A -85,B 0,C 180,E1 -25653.377,E2 -25653.377} C_VEL
LIN {X 0,Y 119.851,Z 775.915,A -85,B 0,C 180,E1 -25660.134,E2 -25660.134} C_VEL
LIN {X 0,Y 121.729,Z 775.994,A -85,B 0,C 180,E1 -25666.78,E2 -25666.78} C_VEL
LIN {X 0,Y 123.217,Z 775.496,A -85,B 0,C 180,E1 -25670.014,E2 -25670.014} C_VEL
LIN {X 0,Y 127.625,Z 773.365,A -85,B 0,C 180,E1 -25676.14,E2 -25676.14} C_VEL
LIN {X 0,Y 133.331,Z 769.751,A -85,B 0,C 180,E1 -25681.812,E2 -25681.812} C_VEL
LIN {X 0,Y 138.199,Z 766.103,A -85,B 0,C 180,E1 -25685.612,E2 -25685.612} C_VEL
LIN {X 0,Y 144.175,Z 761.197,A -85,B 0,C 180,E1 -25689.325,E2 -25689.325} C_VEL
LIN {X 0,Y 151.653,Z 754.255,A -85,B 0,C 180,E1 -25693.123,E2 -25693.123} C_VEL
LIN {X 0,Y 153.716,Z 751.965,A -85,B 0,C 180,E1 -25694.207,E2 -25694.207} C_VEL
LIN {X 0,Y 157.32,Z 746.286,A -85,B 0,C 180,E1 -25697.382,E2 -25697.382} C_VEL
LIN {X 0,Y 158.727,Z 743.742,A -85,B 0,C 180,E1 -25698.827,E2 -25698.827} C_VEL
LIN {X 0,Y 159.805,Z 740.796,A -85,B 0,C 180,E1 -25700.789,E2 -25700.789} C_VEL
LIN {X 0,Y 160.301,Z 737.494,A -85,B 0,C 180,E1 -25703.669,E2 -25703.669} C_VEL
LIN {X 0,Y 160.484,Z 735.048,A -85,B 0,C 180,E1 -25706.312,E2 -25706.312} C_VEL
LIN {X 0,Y 160.527,Z 731.972,A -85,B 0,C 180,E1 -25710.609,E2 -25710.609} C_VEL
LIN {X 0,Y 160.717,Z 730.185,A -85,B 0,C 180,E1 -25714.069,E2 -25714.069} C_VEL
LIN {X 0,Y 160.796,Z 729.279,A -85,B 0,C 180,E1 -25719.533,E2 -25719.533} C_VEL
LIN {X 0,Y 160.958,Z 729.275,A -85,B 0,C 180,E1 -25721.202,E2 -25721.202} C_VEL
LIN {X 0,Y 160.886,Z 729.639,A -85,B 0,C 180,E1 -25722.591,E2 -25722.591} C_VEL
LIN {X 0,Y 160.041,Z 731.205,A -85,B 0,C 180,E1 -25724.609,E2 -25724.609} C_VEL
LIN {X 0,Y 156.248,Z 737.989,A -85,B 0,C 180,E1 -25730.581,E2 -25730.581} C_VEL
LIN {X 0,Y 155.993,Z 739.14,A -85,B 0,C 180,E1 -25732.005,E2 -25732.005} C_VEL
LIN {X 0,Y 155.328,Z 741.689,A -85,B 0,C 180,E1 -25734.808,E2 -25734.808} C_VEL
LIN {X 0,Y 154.775,Z 743.143,A -85,B 0,C 180,E1 -25736.093,E2 -25736.093} C_VEL
LIN {X 0,Y 152.915,Z 746.51,A -85,B 0,C 180,E1 -25738.683,E2 -25738.683} C_VEL
LIN {X 0,Y 151.935,Z 747.65,A -85,B 0,C 180,E1 -25739.338,E2 -25739.338} C_VEL
LIN {X 0,Y 144.093,Z 754.622,A -85,B 0,C 180,E1 -25742.796,E2 -25742.796} C_VEL
LIN {X 0,Y 136.527,Z 760.399,A -85,B 0,C 180,E1 -25746.874,E2 -25746.874} C_VEL
LIN {X 0,Y 131.131,Z 763.922,A -85,B 0,C 180,E1 -25750.495,E2 -25750.495} C_VEL
LIN {X 0,Y 124.39,Z 767.543,A -85,B 0,C 180,E1 -25756.156,E2 -25756.156} C_VEL
LIN {X 0,Y 120.26,Z 769.234,A -85,B 0,C 180,E1 -25760.763,E2 -25760.763} C_VEL
LIN {X 0,Y 116.931,Z 770.052,A -85,B 0,C 180,E1 -25765.634,E2 -25765.634} C_VEL
LIN {X 0,Y 114.463,Z 770.038,A -85,B 0,C 180,E1 -25770.727,E2 -25770.727} C_VEL
LIN {X 0,Y 112.821,Z 769.227,A -85,B 0,C 180,E1 -25775.92,E2 -25775.92} C_VEL
LIN {X 0,Y 111.925,Z 767.64,A -85,B 0,C 180,E1 -25781.103,E2 -25781.103} C_VEL
LIN {X 0,Y 111.745,Z 765.274,A -85,B 0,C 180,E1 -25786.224,E2 -25786.224} C_VEL
LIN {X 0,Y 112.489,Z 760.903,A -85,B 0,C 180,E1 -25792.819,E2 -25792.819} C_VEL
LIN {X 0,Y 113.584,Z 756.35,A -85,B 0,C 180,E1 -25797.936,E2 -25797.936} C_VEL
LIN {X 0,Y 115.707,Z 749.456,A -85,B 0,C 180,E1 -25803.872,E2 -25803.872} C_VEL
LIN {X 0,Y 118.548,Z 741.401,A -85,B 0,C 180,E1 -25809.162,E2 -25809.162} C_VEL
LIN {X 0,Y 121.906,Z 732.058,A -85,B 0,C 180,E1 -25813.828,E2 -25813.828} C_VEL
LIN {X 0,Y 125.179,Z 722.773,A -85,B 0,C 180,E1 -25817.433,E2 -25817.433} C_VEL
LIN {X 0,Y 126.532,Z 718.631,A -85,B 0,C 180,E1 -25818.789,E2 -25818.789} C_VEL
LIN {X 0,Y 126.116,Z 709.583,A -85,B 0,C 180,E1 -25821.99,E2 -25821.99} C_VEL
LIN {X 0,Y 124.971,Z 698.067,A -85,B 0,C 180,E1 -25825.579,E2 -25825.579} C_VEL
LIN {X 0,Y 123.361,Z 688.1,A -85,B 0,C 180,E1 -25828.365,E2 -25828.365} C_VEL
LIN {X 0,Y 121.911,Z 684.251,A -85,B 0,C 180,E1 -25829.671,E2 -25829.671} C_VEL
LIN {X 0,Y 124.62,Z 691.895,A -85,B 0,C 180,E1 -25832.09,E2 -25832.09} C_VEL
LIN {X 0,Y 125.829,Z 702.879,A -85,B 0,C 180,E1 -25835.206,E2 -25835.206} C_VEL
LIN {X 0,Y 126.487,Z 713.915,A -85,B 0,C 180,E1 -25838.788,E2 -25838.788} C_VEL
LIN {X 0,Y 126.401,Z 718.491,A -85,B 0,C 180,E1 -25840.409,E2 -25840.409} C_VEL
LIN {X 0,Y 122.643,Z 729.455,A -85,B 0,C 180,E1 -25844.362,E2 -25844.362} C_VEL
LIN {X 0,Y 119.377,Z 738.489,A -85,B 0,C 180,E1 -25848.596,E2 -25848.596} C_VEL
LIN {X 0,Y 116.348,Z 747.021,A -85,B 0,C 180,E1 -25853.824,E2 -25853.824} C_VEL
LIN {X 0,Y 114.017,Z 754.159,A -85,B 0,C 180,E1 -25859.544,E2 -25859.544} C_VEL
LIN {X 0,Y 112.469,Z 759.859,A -85,B 0,C 180,E1 -25865.674,E2 -25865.674} C_VEL
LIN {X 0,Y 111.72,Z 763.561,A -85,B 0,C 180,E1 -25870.984,E2 -25870.984} C_VEL
LIN {X 0,Y 111.673,Z 766.239,A -85,B 0,C 180,E1 -25876.189,E2 -25876.189} C_VEL
LIN {X 0,Y 112.299,Z 768.04,A -85,B 0,C 180,E1 -25881.256,E2 -25881.256} C_VEL
LIN {X 0,Y 113.564,Z 769.025,A -85,B 0,C 180,E1 -25886.153,E2 -25886.153} C_VEL
LIN {X 0,Y 115.482,Z 769.309,A -85,B 0,C 180,E1 -25890.865,E2 -25890.865} C_VEL
LIN {X 0,Y 118.051,Z 768.933,A -85,B 0,C 180,E1 -25895.371,E2 -25895.371} C_VEL
LIN {X 0,Y 121.23,Z 767.848,A -85,B 0,C 180,E1 -25899.645,E2 -25899.645} C_VEL
LIN {X 0,Y 127.213,Z 764.976,A -85,B 0,C 180,E1 -25905.605,E2 -25905.605} C_VEL
LIN {X 0,Y 134.422,Z 760.438,A -85,B 0,C 180,E1 -25910.976,E2 -25910.976} C_VEL
LIN {X 0,Y 141.118,Z 755.447,A -85,B 0,C 180,E1 -25914.886,E2 -25914.886} C_VEL
LIN {X 0,Y 148.744,Z 748.742,A -85,B 0,C 180,E1 -25918.585,E2 -25918.585} C_VEL
LIN {X 0,Y 152.164,Z 745.412,A -85,B 0,C 180,E1 -25920,E2 -25920} C_VEL
LIN {X 0,Y 153.328,Z 744.002,A -85,B 0,C 180,E1 -25920.722,E2 -25920.722} C_VEL
LIN {X 0,Y 154.998,Z 741.167,A -85,B 0,C 180,E1 -25922.599,E2 -25922.599} C_VEL
LIN {X 0,Y 156.228,Z 738.037,A -85,B 0,C 180,E1 -25925.162,E2 -25925.162} C_VEL
LIN {X 0,Y 156.838,Z 735.513,A -85,B 0,C 180,E1 -25927.726,E2 -25927.726} C_VEL
LIN {X 0,Y 157.055,Z 733.555,A -85,B 0,C 180,E1 -25930.311,E2 -25930.311} C_VEL
LIN {X 0,Y 157.307,Z 730.714,A -85,B 0,C 180,E1 -25935.549,E2 -25935.549} C_VEL
LIN {X 0,Y 156.966,Z 730.226,A -85,B 0,C 180,E1 -25940.989,E2 -25940.989} C_VEL
LIN {X 0,Y 157.059,Z 730.437,A -85,B 0,C 180,E1 -25943.749,E2 -25943.749} C_VEL
LIN {X 0,Y 157.165,Z 731.16,A -85,B 0,C 180,E1 -25946.579,E2 -25946.579} C_VEL
LIN {X 0,Y 157.334,Z 732.314,A -85,B 0,C 180,E1 -25949.43,E2 -25949.43} C_VEL
LIN {X 0,Y 157.459,Z 734.163,A -85,B 0,C 180,E1 -25952.385,E2 -25952.385} C_VEL
LIN {X 0,Y 157.274,Z 736.863,A -85,B 0,C 180,E1 -25955.515,E2 -25955.515} C_VEL
LIN {X 0,Y 156.945,Z 738.488,A -85,B 0,C 180,E1 -25956.958,E2 -25956.958} C_VEL
LIN {X 0,Y 155.353,Z 741.467,A -85,B 0,C 180,E1 -25958.717,E2 -25958.717} C_VEL
LIN {X 0,Y 151.211,Z 747.669,A -85,B 0,C 180,E1 -25961.959,E2 -25961.959} C_VEL
LIN {X 0,Y 147.649,Z 752.184,A -85,B 0,C 180,E1 -25964.442,E2 -25964.442} C_VEL
LIN {X 0,Y 140.988,Z 758.402,A -85,B 0,C 180,E1 -25967.707,E2 -25967.707} C_VEL
LIN {X 0,Y 134.638,Z 763.485,A -85,B 0,C 180,E1 -25971.217,E2 -25971.217} C_VEL
LIN {X 0,Y 129.343,Z 767.237,A -85,B 0,C 180,E1 -25974.793,E2 -25974.793} C_VEL
LIN {X 0,Y 124.112,Z 770.581,A -85,B 0,C 180,E1 -25979.362,E2 -25979.362} C_VEL
LIN {X 0,Y 118.665,Z 773.366,A -85,B 0,C 180,E1 -25985.509,E2 -25985.509} C_VEL
LIN {X 0,Y 114.912,Z 774.617,A -85,B 0,C 180,E1 -25992.195,E2 -25992.195} C_VEL
LIN {X 0,Y 112.845,Z 774.437,A -85,B 0,C 180,E1 -25999.233,E2 -25999.233} C_VEL
LIN {X 0,Y 112.402,Z 773.8,A -85,B 0,C 180,E1 -26002.818,E2 -26002.818} C_VEL
LIN {X 0,Y 112.401,Z 771.944,A -85,B 0,C 180,E1 -26009.106,E2 -26009.106} C_VEL
LIN {X 0,Y 112.3,Z 773.834,A -85,B 0,C 180,E1 -26013.59,E2 -26013.59} C_VEL
LIN {X 0,Y 112.405,Z 774.908,A -85,B 0,C 180,E1 -26017.185,E2 -26017.185} C_VEL
LIN {X 0,Y 113.7,Z 775.878,A -85,B 0,C 180,E1 -26024.316,E2 -26024.316} C_VEL
LIN {X 0,Y 116.547,Z 775.408,A -85,B 0,C 180,E1 -26031.213,E2 -26031.213} C_VEL
LIN {X 0,Y 121.299,Z 773.524,A -85,B 0,C 180,E1 -26037.616,E2 -26037.616} C_VEL
LIN {X 0,Y 127.356,Z 770.1,A -85,B 0,C 180,E1 -26043.495,E2 -26043.495} C_VEL
LIN {X 0,Y 132.521,Z 766.676,A -85,B 0,C 180,E1 -26047.391,E2 -26047.391} C_VEL
LIN {X 0,Y 138.806,Z 761.99,A -85,B 0,C 180,E1 -26051.165,E2 -26051.165} C_VEL
LIN {X 0,Y 146.608,Z 755.278,A -85,B 0,C 180,E1 -26054.999,E2 -26054.999} C_VEL
LIN {X 0,Y 147.787,Z 754.208,A -85,B 0,C 180,E1 -26055.507,E2 -26055.507} C_VEL
LIN {X 0,Y 151.131,Z 749.917,A -85,B 0,C 180,E1 -26058.078,E2 -26058.078} C_VEL
LIN {X 0,Y 153.202,Z 746.736,A -85,B 0,C 180,E1 -26060.041,E2 -26060.041} C_VEL
LIN {X 0,Y 153.869,Z 745.404,A -85,B 0,C 180,E1 -26060.941,E2 -26060.941} C_VEL
LIN {X 0,Y 154.343,Z 744.073,A -85,B 0,C 180,E1 -26062.029,E2 -26062.029} C_VEL
LIN {X 0,Y 154.952,Z 741.384,A -85,B 0,C 180,E1 -26064.728,E2 -26064.728} C_VEL
LIN {X 0,Y 155.234,Z 739.411,A -85,B 0,C 180,E1 -26067.093,E2 -26067.093} C_VEL
LIN {X 0,Y 155.439,Z 737.369,A -85,B 0,C 180,E1 -26070.175,E2 -26070.175} C_VEL
LIN {X 0,Y 155.818,Z 735.251,A -85,B 0,C 180,E1 -26074.434,E2 -26074.434} C_VEL
LIN {X 0,Y 155.883,Z 734.515,A -85,B 0,C 180,E1 -26078.858,E2 -26078.858} C_VEL
LIN {X 0,Y 156.166,Z 734.439,A -85,B 0,C 180,E1 -26081.638,E2 -26081.638} C_VEL
LIN {X 0,Y 156.19,Z 735.036,A -85,B 0,C 180,E1 -26084.337,E2 -26084.337} C_VEL
LIN {X 0,Y 156.215,Z 736.065,A -85,B 0,C 180,E1 -26087,E2 -26087} C_VEL
LIN {X 0,Y 156.151,Z 737.496,A -85,B 0,C 180,E1 -26089.629,E2 -26089.629} C_VEL
LIN {X 0,Y 155.993,Z 739.14,A -85,B 0,C 180,E1 -26092.005,E2 -26092.005} C_VEL
LIN {X 0,Y 155.494,Z 740.491,A -85,B 0,C 180,E1 -26093.335,E2 -26093.335} C_VEL
LIN {X 0,Y 153.84,Z 742.866,A -85,B 0,C 180,E1 -26094.808,E2 -26094.808} C_VEL
LIN {X 0,Y 151.413,Z 745.605,A -85,B 0,C 180,E1 -26096.1,E2 -26096.1} C_VEL
LIN {X 0,Y 145.067,Z 751.285,A -85,B 0,C 180,E1 -26098.465,E2 -26098.465} C_VEL
LIN {X 0,Y 139.758,Z 755.422,A -85,B 0,C 180,E1 -26100.522,E2 -26100.522} C_VEL
LIN {X 0,Y 131.533,Z 761.153,A -85,B 0,C 180,E1 -26104.724,E2 -26104.724} C_VEL
LIN {X 0,Y 123.868,Z 765.6,A -85,B 0,C 180,E1 -26109.8,E2 -26109.8} C_VEL
LIN {X 0,Y 116.894,Z 768.707,A -85,B 0,C 180,E1 -26115.849,E2 -26115.849} C_VEL
LIN {X 0,Y 111.718,Z 770.147,A -85,B 0,C 180,E1 -26122.176,E2 -26122.176} C_VEL
LIN {X 0,Y 108.94,Z 770.394,A -85,B 0,C 180,E1 -26126.846,E2 -26126.846} C_VEL
LIN {X 0,Y 106.835,Z 769.933,A -85,B 0,C 180,E1 -26131.754,E2 -26131.754} C_VEL
LIN {X 0,Y 105.475,Z 768.81,A -85,B 0,C 180,E1 -26136.908,E2 -26136.908} C_VEL
LIN {X 0,Y 104.721,Z 766.869,A -85,B 0,C 180,E1 -26142.417,E2 -26142.417} C_VEL
LIN {X 0,Y 104.75,Z 764.118,A -85,B 0,C 180,E1 -26147.859,E2 -26147.859} C_VEL
LIN {X 0,Y 105.665,Z 759.613,A -85,B 0,C 180,E1 -26154.408,E2 -26154.408} C_VEL
LIN {X 0,Y 107.314,Z 753.488,A -85,B 0,C 180,E1 -26160.927,E2 -26160.927} C_VEL
LIN {X 0,Y 109.485,Z 747.153,A -85,B 0,C 180,E1 -26166.122,E2 -26166.122} C_VEL
LIN {X 0,Y 112.378,Z 739.363,A -85,B 0,C 180,E1 -26171.13,E2 -26171.13} C_VEL
LIN {X 0,Y 115.953,Z 729.797,A -85,B 0,C 180,E1 -26175.877,E2 -26175.877} C_VEL
LIN {X 0,Y 119.763,Z 719.205,A -85,B 0,C 180,E1 -26179.859,E2 -26179.859} C_VEL
LIN {X 0,Y 119.34,Z 709.035,A -85,B 0,C 180,E1 -26183.659,E2 -26183.659} C_VEL
LIN {X 0,Y 118.42,Z 698.873,A -85,B 0,C 180,E1 -26187.022,E2 -26187.022} C_VEL
LIN {X 0,Y 117.085,Z 690.59,A -85,B 0,C 180,E1 -26189.568,E2 -26189.568} C_VEL
LIN {X 0,Y 118.23,Z 693.991,A -85,B 0,C 180,E1 -26190.851,E2 -26190.851} C_VEL
LIN {X 0,Y 119.27,Z 703.452,A -85,B 0,C 180,E1 -26193.8,E2 -26193.8} C_VEL
LIN {X 0,Y 119.797,Z 714.36,A -85,B 0,C 180,E1 -26197.584,E2 -26197.584} C_VEL
LIN {X 0,Y 119.676,Z 718.897,A -85,B 0,C 180,E1 -26199.292,E2 -26199.292} C_VEL
LIN {X 0,Y 115.675,Z 730.108,A -85,B 0,C 180,E1 -26203.564,E2 -26203.564} C_VEL
LIN {X 0,Y 112.116,Z 739.434,A -85,B 0,C 180,E1 -26208.264,E2 -26208.264} C_VEL
LIN {X 0,Y 109.085,Z 747.792,A -85,B 0,C 180,E1 -26213.792,E2 -26213.792} C_VEL
LIN {X 0,Y 107.002,Z 753.899,A -85,B 0,C 180,E1 -26219.01,E2 -26219.01} C_VEL
LIN {X 0,Y 105.626,Z 758.736,A -85,B 0,C 180,E1 -26224.287,E2 -26224.287} C_VEL
LIN {X 0,Y 104.729,Z 762.519,A -85,B 0,C 180,E1 -26229.604,E2 -26229.604} C_VEL
LIN {X 0,Y 104.532,Z 765.396,A -85,B 0,C 180,E1 -26234.9,E2 -26234.9} C_VEL
LIN {X 0,Y 104.703,Z 766.65,A -85,B 0,C 180,E1 -26237.837,E2 -26237.837} C_VEL
LIN {X 0,Y 105.559,Z 768.363,A -85,B 0,C 180,E1 -26243.187,E2 -26243.187} C_VEL
LIN {X 0,Y 107.175,Z 769.326,A -85,B 0,C 180,E1 -26248.478,E2 -26248.478} C_VEL
LIN {X 0,Y 109.679,Z 769.511,A -85,B 0,C 180,E1 -26253.774,E2 -26253.774} C_VEL
LIN {X 0,Y 113.024,Z 768.91,A -85,B 0,C 180,E1 -26258.858,E2 -26258.858} C_VEL
LIN {X 0,Y 117.185,Z 767.502,A -85,B 0,C 180,E1 -26263.646,E2 -26263.646} C_VEL
LIN {X 0,Y 122.115,Z 765.271,A -85,B 0,C 180,E1 -26268.058,E2 -26268.058} C_VEL
LIN {X 0,Y 127.716,Z 762.175,A -85,B 0,C 180,E1 -26272.087,E2 -26272.087} C_VEL
LIN {X 0,Y 133.893,Z 758.117,A -85,B 0,C 180,E1 -26275.767,E2 -26275.767} C_VEL
LIN {X 0,Y 140.575,Z 753.044,A -85,B 0,C 180,E1 -26279.065,E2 -26279.065} C_VEL
LIN {X 0,Y 147.68,Z 746.85,A -85,B 0,C 180,E1 -26282.066,E2 -26282.066} C_VEL
LIN {X 0,Y 149.661,Z 744.074,A -85,B 0,C 180,E1 -26284.039,E2 -26284.039} C_VEL
LIN {X 0,Y 150.973,Z 741.26,A -85,B 0,C 180,E1 -26286.683,E2 -26286.683} C_VEL
LIN {X 0,Y 151.373,Z 740.138,A -85,B 0,C 180,E1 -26288.006,E2 -26288.006} C_VEL
LIN {X 0,Y 151.778,Z 738.239,A -85,B 0,C 180,E1 -26290.674,E2 -26290.674} C_VEL
LIN {X 0,Y 152.104,Z 736.522,A -85,B 0,C 180,E1 -26294.002,E2 -26294.002} C_VEL
LIN {X 0,Y 152.256,Z 735.699,A -85,B 0,C 180,E1 -26296.079,E2 -26296.079} C_VEL
LIN {X 0,Y 152.045,Z 735.385,A -85,B 0,C 180,E1 -26301.702,E2 -26301.702} C_VEL
LIN {X 0,Y 152.112,Z 735.727,A -85,B 0,C 180,E1 -26304.571,E2 -26304.571} C_VEL
LIN {X 0,Y 152.243,Z 737.055,A -85,B 0,C 180,E1 -26308.708,E2 -26308.708} C_VEL
LIN {X 0,Y 152.245,Z 738.925,A -85,B 0,C 180,E1 -26312.07,E2 -26312.07} C_VEL
LIN {X 0,Y 151.9,Z 741.016,A -85,B 0,C 180,E1 -26314.75,E2 -26314.75} C_VEL
LIN {X 0,Y 151.436,Z 742.427,A -85,B 0,C 180,E1 -26316.047,E2 -26316.047} C_VEL
LIN {X 0,Y 148.688,Z 746.386,A -85,B 0,C 180,E1 -26318.391,E2 -26318.391} C_VEL
LIN {X 0,Y 142.791,Z 753.376,A -85,B 0,C 180,E1 -26322.417,E2 -26322.417} C_VEL
LIN {X 0,Y 135.866,Z 759.289,A -85,B 0,C 180,E1 -26325.709,E2 -26325.709} C_VEL
LIN {X 0,Y 127.108,Z 765.511,A -85,B 0,C 180,E1 -26330.519,E2 -26330.519} C_VEL
LIN {X 0,Y 121.417,Z 769.012,A -85,B 0,C 180,E1 -26334.633,E2 -26334.633} C_VEL
LIN {X 0,Y 114.981,Z 772.314,A -85,B 0,C 180,E1 -26340.728,E2 -26340.728} C_VEL
LIN {X 0,Y 109.909,Z 774.096,A -85,B 0,C 180,E1 -26347.441,E2 -26347.441} C_VEL
LIN {X 0,Y 106.791,Z 774.465,A -85,B 0,C 180,E1 -26354.739,E2 -26354.739} C_VEL
LIN {X 0,Y 105.363,Z 773.336,A -85,B 0,C 180,E1 -26362.335,E2 -26362.335} C_VEL
LIN {X 0,Y 105.345,Z 771.266,A -85,B 0,C 180,E1 -26369.046,E2 -26369.046} C_VEL
LIN {X 0,Y 105.225,Z 773.268,A -85,B 0,C 180,E1 -26373.831,E2 -26373.831} C_VEL
LIN {X 0,Y 105.894,Z 775.191,A -85,B 0,C 180,E1 -26381.486,E2 -26381.486} C_VEL
LIN {X 0,Y 108.15,Z 775.644,A -85,B 0,C 180,E1 -26388.962,E2 -26388.962} C_VEL
LIN {X 0,Y 112.284,Z 774.643,A -85,B 0,C 180,E1 -26395.987,E2 -26395.987} C_VEL
LIN {X 0,Y 118.098,Z 772.245,A -85,B 0,C 180,E1 -26402.385,E2 -26402.385} C_VEL
LIN {X 0,Y 123.873,Z 769.115,A -85,B 0,C 180,E1 -26407.193,E2 -26407.193} C_VEL
LIN {X 0,Y 131.359,Z 764.302,A -85,B 0,C 180,E1 -26411.974,E2 -26411.974} C_VEL
LIN {X 0,Y 138.171,Z 759.304,A -85,B 0,C 180,E1 -26415.408,E2 -26415.408} C_VEL
LIN {X 0,Y 142.911,Z 755.34,A -85,B 0,C 180,E1 -26417.534,E2 -26417.534} C_VEL
LIN {X 0,Y 146.354,Z 751.272,A -85,B 0,C 180,E1 -26420.206,E2 -26420.206} C_VEL
LIN {X 0,Y 148.149,Z 748.768,A -85,B 0,C 180,E1 -26421.924,E2 -26421.924} C_VEL
LIN {X 0,Y 148.842,Z 747.24,A -85,B 0,C 180,E1 -26423.391,E2 -26423.391} C_VEL
LIN {X 0,Y 149.443,Z 745.248,A -85,B 0,C 180,E1 -26425.644,E2 -26425.644} C_VEL
LIN {X 0,Y 149.963,Z 742.916,A -85,B 0,C 180,E1 -26428.968,E2 -26428.968} C_VEL
LIN {X 0,Y 150.333,Z 740.964,A -85,B 0,C 180,E1 -26432.655,E2 -26432.655} C_VEL
LIN {X 0,Y 150.641,Z 740.009,A -85,B 0,C 180,E1 -26435.173,E2 -26435.173} C_VEL
LIN {X 0,Y 150.959,Z 739.353,A -85,B 0,C 180,E1 -26440.981,E2 -26440.981} C_VEL
LIN {X 0,Y 150.978,Z 739.766,A -85,B 0,C 180,E1 -26443.782,E2 -26443.782} C_VEL
LIN {X 0,Y 150.937,Z 740.689,A -85,B 0,C 180,E1 -26446.537,E2 -26446.537} C_VEL
LIN {X 0,Y 150.716,Z 741.964,A -85,B 0,C 180,E1 -26449.25,E2 -26449.25} C_VEL
LIN {X 0,Y 150.413,Z 743.675,A -85,B 0,C 180,E1 -26451.942,E2 -26451.942} C_VEL
LIN {X 0,Y 149.414,Z 745.971,A -85,B 0,C 180,E1 -26454.602,E2 -26454.602} C_VEL
LIN {X 0,Y 147.372,Z 749.096,A -85,B 0,C 180,E1 -26457.267,E2 -26457.267} C_VEL
LIN {X 0,Y 139.758,Z 755.422,A -85,B 0,C 180,E1 -26460.522,E2 -26460.522} C_VEL
LIN {X 0,Y 135.818,Z 758.117,A -85,B 0,C 180,E1 -26461.978,E2 -26461.978} C_VEL
LIN {X 0,Y 128.194,Z 762.159,A -85,B 0,C 180,E1 -26464.112,E2 -26464.112} C_VEL
LIN {X 0,Y 120.653,Z 765.438,A -85,B 0,C 180,E1 -26466.637,E2 -26466.637} C_VEL
LIN {X 0,Y 116.953,Z 766.937,A -85,B 0,C 180,E1 -26468.723,E2 -26468.723} C_VEL
LIN {X 0,Y 109.393,Z 769.667,A -85,B 0,C 180,E1 -26475.485,E2 -26475.485} C_VEL
LIN {X 0,Y 105.187,Z 770.504,A -85,B 0,C 180,E1 -26480.704,E2 -26480.704} C_VEL
LIN {X 0,Y 101.886,Z 770.533,A -85,B 0,C 180,E1 -26486.266,E2 -26486.266} C_VEL
LIN {X 0,Y 98.789,Z 769.195,A -85,B 0,C 180,E1 -26494.69,E2 -26494.69} C_VEL
LIN {X 0,Y 97.809,Z 767.401,A -85,B 0,C 180,E1 -26500.293,E2 -26500.293} C_VEL
LIN {X 0,Y 97.672,Z 763.828,A -85,B 0,C 180,E1 -26507.923,E2 -26507.923} C_VEL
LIN {X 0,Y 98.72,Z 758.86,A -85,B 0,C 180,E1 -26515.281,E2 -26515.281} C_VEL
LIN {X 0,Y 100.712,Z 752.155,A -85,B 0,C 180,E1 -26522.583,E2 -26522.583} C_VEL
LIN {X 0,Y 103.088,Z 745.613,A -85,B 0,C 180,E1 -26527.976,E2 -26527.976} C_VEL
LIN {X 0,Y 106.631,Z 736.481,A -85,B 0,C 180,E1 -26533.731,E2 -26533.731} C_VEL
LIN {X 0,Y 110.64,Z 726.325,A -85,B 0,C 180,E1 -26538.563,E2 -26538.563} C_VEL
LIN {X 0,Y 113.048,Z 719.695,A -85,B 0,C 180,E1 -26541.057,E2 -26541.057} C_VEL
LIN {X 0,Y 112.669,Z 708.478,A -85,B 0,C 180,E1 -26545.527,E2 -26545.527} C_VEL
LIN {X 0,Y 111.765,Z 698.321,A -85,B 0,C 180,E1 -26549.098,E2 -26549.098} C_VEL
LIN {X 0,Y 111.601,Z 696.653,A -85,B 0,C 180,E1 -26549.66,E2 -26549.66} C_VEL
LIN {X 0,Y 112.118,Z 697.276,A -85,B 0,C 180,E1 -26549.998,E2 -26549.998} C_VEL
LIN {X 0,Y 112.905,Z 707.762,A -85,B 0,C 180,E1 -26553.567,E2 -26553.567} C_VEL
LIN {X 0,Y 113.133,Z 718.167,A -85,B 0,C 180,E1 -26557.584,E2 -26557.584} C_VEL
LIN {X 0,Y 112.53,Z 720.654,A -85,B 0,C 180,E1 -26558.529,E2 -26558.529} C_VEL
LIN {X 0,Y 108.719,Z 730.818,A -85,B 0,C 180,E1 -26562.696,E2 -26562.696} C_VEL
LIN {X 0,Y 105.097,Z 739.749,A -85,B 0,C 180,E1 -26567.511,E2 -26567.511} C_VEL
LIN {X 0,Y 101.999,Z 747.987,A -85,B 0,C 180,E1 -26573.338,E2 -26573.338} C_VEL
LIN {X 0,Y 99.616,Z 754.718,A -85,B 0,C 180,E1 -26579.592,E2 -26579.592} C_VEL
LIN {X 0,Y 98.102,Z 760.159,A -85,B 0,C 180,E1 -26586.315,E2 -26586.315} C_VEL
LIN {X 0,Y 97.439,Z 764.612,A -85,B 0,C 180,E1 -26593.84,E2 -26593.84} C_VEL
LIN {X 0,Y 98.154,Z 767.786,A -85,B 0,C 180,E1 -26601.96,E2 -26601.96} C_VEL
LIN {X 0,Y 99.679,Z 769.165,A -85,B 0,C 180,E1 -26607.783,E2 -26607.783} C_VEL
LIN {X 0,Y 102.133,Z 769.741,A -85,B 0,C 180,E1 -26613.448,E2 -26613.448} C_VEL
LIN {X 0,Y 106.896,Z 769.259,A -85,B 0,C 180,E1 -26620.808,E2 -26620.808} C_VEL
LIN {X 0,Y 110.95,Z 768.127,A -85,B 0,C 180,E1 -26625.322,E2 -26625.322} C_VEL
LIN {X 0,Y 118.163,Z 765.162,A -85,B 0,C 180,E1 -26631.363,E2 -26631.363} C_VEL
LIN {X 0,Y 126.872,Z 760.444,A -85,B 0,C 180,E1 -26636.824,E2 -26636.824} C_VEL
LIN {X 0,Y 135.091,Z 754.91,A -85,B 0,C 180,E1 -26640.871,E2 -26640.871} C_VEL
LIN {X 0,Y 142.31,Z 749.213,A -85,B 0,C 180,E1 -26643.796,E2 -26643.796} C_VEL
LIN {X 0,Y 143.255,Z 748.253,A -85,B 0,C 180,E1 -26644.39,E2 -26644.39} C_VEL
LIN {X 0,Y 144.321,Z 746.882,A -85,B 0,C 180,E1 -26645.589,E2 -26645.589} C_VEL
LIN {X 0,Y 145.666,Z 744.461,A -85,B 0,C 180,E1 -26648.322,E2 -26648.322} C_VEL
LIN {X 0,Y 146.314,Z 742.661,A -85,B 0,C 180,E1 -26651.077,E2 -26651.077} C_VEL
LIN {X 0,Y 146.752,Z 741.327,A -85,B 0,C 180,E1 -26653.854,E2 -26653.854} C_VEL
LIN {X 0,Y 146.951,Z 740.416,A -85,B 0,C 180,E1 -26656.965,E2 -26656.965} C_VEL
LIN {X 0,Y 146.866,Z 740.308,A -85,B 0,C 180,E1 -26662.509,E2 -26662.509} C_VEL
LIN {X 0,Y 146.874,Z 740.83,A -85,B 0,C 180,E1 -26665.509,E2 -26665.509} C_VEL
LIN {X 0,Y 146.947,Z 741.797,A -85,B 0,C 180,E1 -26668.572,E2 -26668.572} C_VEL
LIN {X 0,Y 146.758,Z 743.438,A -85,B 0,C 180,E1 -26671.788,E2 -26671.788} C_VEL
LIN {X 0,Y 146.398,Z 744.881,A -85,B 0,C 180,E1 -26673.83,E2 -26673.83} C_VEL
LIN {X 0,Y 145.81,Z 746.06,A -85,B 0,C 180,E1 -26674.978,E2 -26674.978} C_VEL
LIN {X 0,Y 143.149,Z 749.279,A -85,B 0,C 180,E1 -26676.993,E2 -26676.993} C_VEL
LIN {X 0,Y 138.112,Z 754.495,A -85,B 0,C 180,E1 -26680.247,E2 -26680.247} C_VEL
LIN {X 0,Y 130.923,Z 760.139,A -85,B 0,C 180,E1 -26683.56,E2 -26683.56} C_VEL
LIN {X 0,Y 123.953,Z 764.755,A -85,B 0,C 180,E1 -26687.128,E2 -26687.128} C_VEL
LIN {X 0,Y 119.112,Z 767.582,A -85,B 0,C 180,E1 -26690.089,E2 -26690.089} C_VEL
LIN {X 0,Y 112.106,Z 771.09,A -85,B 0,C 180,E1 -26695.654,E2 -26695.654} C_VEL
LIN {X 0,Y 105.89,Z 773.401,A -85,B 0,C 180,E1 -26702.318,E2 -26702.318} C_VEL
LIN {X 0,Y 101.407,Z 774.285,A -85,B 0,C 180,E1 -26709.727,E2 -26709.727} C_VEL
LIN {X 0,Y 98.897,Z 773.684,A -85,B 0,C 180,E1 -26717.692,E2 -26717.692} C_VEL
LIN {X 0,Y 98.174,Z 771.644,A -85,B 0,C 180,E1 -26725.897,E2 -26725.897} C_VEL
LIN {X 0,Y 98.287,Z 770.519,A -85,B 0,C 180,E1 -26728.977,E2 -26728.977} C_VEL
LIN {X 0,Y 98.174,Z 772.676,A -85,B 0,C 180,E1 -26734.107,E2 -26734.107} C_VEL
LIN {X 0,Y 98.93,Z 774.764,A -85,B 0,C 180,E1 -26742.307,E2 -26742.307} C_VEL
LIN {X 0,Y 101.427,Z 775.42,A -85,B 0,C 180,E1 -26750.272,E2 -26750.272} C_VEL
LIN {X 0,Y 105.938,Z 774.656,A -85,B 0,C 180,E1 -26757.672,E2 -26757.672} C_VEL
LIN {X 0,Y 112.16,Z 772.443,A -85,B 0,C 180,E1 -26764.331,E2 -26764.331} C_VEL
LIN {X 0,Y 119.656,Z 768.797,A -85,B 0,C 180,E1 -26770.249,E2 -26770.249} C_VEL
LIN {X 0,Y 126.208,Z 764.994,A -85,B 0,C 180,E1 -26774.114,E2 -26774.114} C_VEL
LIN {X 0,Y 133.329,Z 760.208,A -85,B 0,C 180,E1 -26777.56,E2 -26777.56} C_VEL
LIN {X 0,Y 138.17,Z 756.477,A -85,B 0,C 180,E1 -26779.729,E2 -26779.729} C_VEL
LIN {X 0,Y 141.786,Z 752.653,A -85,B 0,C 180,E1 -26782.476,E2 -26782.476} C_VEL
LIN {X 0,Y 142.823,Z 751.165,A -85,B 0,C 180,E1 -26783.808,E2 -26783.808} C_VEL
LIN {X 0,Y 143.71,Z 749.168,A -85,B 0,C 180,E1 -26786.241,E2 -26786.241} C_VEL
LIN {X 0,Y 144.003,Z 748.277,A -85,B 0,C 180,E1 -26787.531,E2 -26787.531} C_VEL
LIN {X 0,Y 144.561,Z 746.358,A -85,B 0,C 180,E1 -26791.057,E2 -26791.057} C_VEL
LIN {X 0,Y 145.032,Z 745.044,A -85,B 0,C 180,E1 -26794.143,E2 -26794.143} C_VEL
LIN {X 0,Y 145.264,Z 744.307,A -85,B 0,C 180,E1 -26797.229,E2 -26797.229} C_VEL
LIN {X 0,Y 145.488,Z 744.035,A -85,B 0,C 180,E1 -26800.236,E2 -26800.236} C_VEL
LIN {X 0,Y 145.552,Z 744.268,A -85,B 0,C 180,E1 -26803.159,E2 -26803.159} C_VEL
LIN {X 0,Y 145.425,Z 745.033,A -85,B 0,C 180,E1 -26806.017,E2 -26806.017} C_VEL
LIN {X 0,Y 145.102,Z 746.182,A -85,B 0,C 180,E1 -26808.829,E2 -26808.829} C_VEL
LIN {X 0,Y 144.581,Z 747.794,A -85,B 0,C 180,E1 -26811.615,E2 -26811.615} C_VEL
LIN {X 0,Y 143.988,Z 748.841,A -85,B 0,C 180,E1 -26812.991,E2 -26812.991} C_VEL
LIN {X 0,Y 142.452,Z 750.954,A -85,B 0,C 180,E1 -26815.178,E2 -26815.178} C_VEL
LIN {X 0,Y 139.833,Z 753.142,A -85,B 0,C 180,E1 -26816.401,E2 -26816.401} C_VEL
LIN {X 0,Y 131.472,Z 759.068,A -85,B 0,C 180,E1 -26820,E2 -26820} C_VEL
LIN {X 0,Y 122.692,Z 764.194,A -85,B 0,C 180,E1 -26824.772,E2 -26824.772} C_VEL
LIN {X 0,Y 116.953,Z 766.937,A -85,B 0,C 180,E1 -26828.723,E2 -26828.723} C_VEL
LIN {X 0,Y 113.368,Z 768.24,A -85,B 0,C 180,E1 -26830.985,E2 -26830.985} C_VEL
LIN {X 0,Y 106.356,Z 769.897,A -85,B 0,C 180,E1 -26834.55,E2 -26834.55} C_VEL
LIN {X 0,Y 99.777,Z 770.811,A -85,B 0,C 180,E1 -26838.635,E2 -26838.635} C_VEL
LIN {X 0,Y 97.004,Z 770.832,A -85,B 0,C 180,E1 -26841.667,E2 -26841.667} C_VEL
LIN {X 0,Y 94.35,Z 770.501,A -85,B 0,C 180,E1 -26846.634,E2 -26846.634} C_VEL
LIN {X 0,Y 92.089,Z 769.361,A -85,B 0,C 180,E1 -26852.911,E2 -26852.911} C_VEL
LIN {X 0,Y 90.563,Z 766.495,A -85,B 0,C 180,E1 -26861.672,E2 -26861.672} C_VEL
LIN {X 0,Y 90.629,Z 763.268,A -85,B 0,C 180,E1 -26868.366,E2 -26868.366} C_VEL
LIN {X 0,Y 91.472,Z 759.217,A -85,B 0,C 180,E1 -26874.725,E2 -26874.725} C_VEL
LIN {X 0,Y 93.239,Z 753.218,A -85,B 0,C 180,E1 -26881.892,E2 -26881.892} C_VEL
LIN {X 0,Y 95.99,Z 745.904,A -85,B 0,C 180,E1 -26888.524,E2 -26888.524} C_VEL
LIN {X 0,Y 99.487,Z 737.371,A -85,B 0,C 180,E1 -26894.341,E2 -26894.341} C_VEL
LIN {X 0,Y 103.323,Z 727.992,A -85,B 0,C 180,E1 -26899.217,E2 -26899.217} C_VEL
LIN {X 0,Y 106.316,Z 720.206,A -85,B 0,C 180,E1 -26902.401,E2 -26902.401} C_VEL
LIN {X 0,Y 106.136,Z 710.167,A -85,B 0,C 180,E1 -26906.677,E2 -26906.677} C_VEL
LIN {X 0,Y 105.666,Z 702.499,A -85,B 0,C 180,E1 -26909.641,E2 -26909.641} C_VEL
LIN {X 0,Y 106.174,Z 703.068,A -85,B 0,C 180,E1 -26909.998,E2 -26909.998} C_VEL
LIN {X 0,Y 106.444,Z 714.2,A -85,B 0,C 180,E1 -26914.306,E2 -26914.306} C_VEL
LIN {X 0,Y 106.189,Z 720.217,A -85,B 0,C 180,E1 -26916.895,E2 -26916.895} C_VEL
LIN {X 0,Y 102.003,Z 730.813,A -85,B 0,C 180,E1 -26921.423,E2 -26921.423} C_VEL
LIN {X 0,Y 98.124,Z 739.973,A -85,B 0,C 180,E1 -26926.646,E2 -26926.646} C_VEL
LIN {X 0,Y 94.993,Z 747.922,A -85,B 0,C 180,E1 -26932.629,E2 -26932.629} C_VEL
LIN {X 0,Y 92.435,Z 754.952,A -85,B 0,C 180,E1 -26939.615,E2 -26939.615} C_VEL
LIN {X 0,Y 91.137,Z 759.38,A -85,B 0,C 180,E1 -26945.33,E2 -26945.33} C_VEL
LIN {X 0,Y 90.395,Z 763.15,A -85,B 0,C 180,E1 -26951.6,E2 -26951.6} C_VEL
LIN {X 0,Y 90.373,Z 765.083,A -85,B 0,C 180,E1 -26955.581,E2 -26955.581} C_VEL
LIN {X 0,Y 91.008,Z 767.424,A -85,B 0,C 180,E1 -26961.844,E2 -26961.844} C_VEL
LIN {X 0,Y 92.464,Z 768.972,A -85,B 0,C 180,E1 -26967.855,E2 -26967.855} C_VEL
LIN {X 0,Y 94.82,Z 769.825,A -85,B 0,C 180,E1 -26973.594,E2 -26973.594} C_VEL
LIN {X 0,Y 97.923,Z 769.955,A -85,B 0,C 180,E1 -26978.97,E2 -26978.97} C_VEL
LIN {X 0,Y 102.147,Z 769.351,A -85,B 0,C 180,E1 -26984.408,E2 -26984.408} C_VEL
LIN {X 0,Y 107.247,Z 767.956,A -85,B 0,C 180,E1 -26989.397,E2 -26989.397} C_VEL
LIN {X 0,Y 113.098,Z 765.775,A -85,B 0,C 180,E1 -26993.839,E2 -26993.839} C_VEL
LIN {X 0,Y 121.565,Z 761.632,A -85,B 0,C 180,E1 -26998.935,E2 -26998.935} C_VEL
LIN {X 0,Y 130.414,Z 756.265,A -85,B 0,C 180,E1 -27003.089,E2 -27003.089} C_VEL
LIN {X 0,Y 137.6,Z 751.101,A -85,B 0,C 180,E1 -27005.863,E2 -27005.863} C_VEL
LIN {X 0,Y 138.963,Z 749.628,A -85,B 0,C 180,E1 -27007.264,E2 -27007.264} C_VEL
LIN {X 0,Y 139.74,Z 748.503,A -85,B 0,C 180,E1 -27008.678,E2 -27008.678} C_VEL
LIN {X 0,Y 140.653,Z 746.823,A -85,B 0,C 180,E1 -27011.529,E2 -27011.529} C_VEL
LIN {X 0,Y 141.213,Z 745.577,A -85,B 0,C 180,E1 -27014.409,E2 -27014.409} C_VEL
LIN {X 0,Y 141.469,Z 744.901,A -85,B 0,C 180,E1 -27017.342,E2 -27017.342} C_VEL
LIN {X 0,Y 141.387,Z 744.782,A -85,B 0,C 180,E1 -27020.362,E2 -27020.362} C_VEL
LIN {X 0,Y 141.425,Z 744.993,A -85,B 0,C 180,E1 -27023.425,E2 -27023.425} C_VEL
LIN {X 0,Y 141.35,Z 745.69,A -85,B 0,C 180,E1 -27026.583,E2 -27026.583} C_VEL
LIN {X 0,Y 141.222,Z 746.835,A -85,B 0,C 180,E1 -27029.845,E2 -27029.845} C_VEL
LIN {X 0,Y 140.926,Z 748.018,A -85,B 0,C 180,E1 -27032.03,E2 -27032.03} C_VEL
LIN {X 0,Y 140.51,Z 748.996,A -85,B 0,C 180,E1 -27033.38,E2 -27033.38} C_VEL
LIN {X 0,Y 139.573,Z 750.045,A -85,B 0,C 180,E1 -27034.212,E2 -27034.212} C_VEL
LIN {X 0,Y 133.638,Z 755.669,A -85,B 0,C 180,E1 -27037.925,E2 -27037.925} C_VEL
LIN {X 0,Y 126.18,Z 761.024,A -85,B 0,C 180,E1 -27041.245,E2 -27041.245} C_VEL
LIN {X 0,Y 116.548,Z 766.61,A -85,B 0,C 180,E1 -27046.097,E2 -27046.097} C_VEL
LIN {X 0,Y 110.155,Z 769.721,A -85,B 0,C 180,E1 -27050.359,E2 -27050.359} C_VEL
LIN {X 0,Y 102.791,Z 772.542,A -85,B 0,C 180,E1 -27056.842,E2 -27056.842} C_VEL
LIN {X 0,Y 96.925,Z 773.904,A -85,B 0,C 180,E1 -27064.213,E2 -27064.213} C_VEL
LIN {X 0,Y 93.114,Z 773.831,A -85,B 0,C 180,E1 -27072.43,E2 -27072.43} C_VEL
LIN {X 0,Y 91.295,Z 772.352,A -85,B 0,C 180,E1 -27081.145,E2 -27081.145} C_VEL
LIN {X 0,Y 91.246,Z 769.876,A -85,B 0,C 180,E1 -27089.174,E2 -27089.174} C_VEL
LIN {X 0,Y 91.117,Z 772.013,A -85,B 0,C 180,E1 -27094.426,E2 -27094.426} C_VEL
LIN {X 0,Y 92.002,Z 774.332,A -85,B 0,C 180,E1 -27103.25,E2 -27103.25} C_VEL
LIN {X 0,Y 94.768,Z 775.158,A -85,B 0,C 180,E1 -27111.767,E2 -27111.767} C_VEL
LIN {X 0,Y 99.698,Z 774.612,A -85,B 0,C 180,E1 -27119.569,E2 -27119.569} C_VEL
LIN {X 0,Y 106.369,Z 772.658,A -85,B 0,C 180,E1 -27126.489,E2 -27126.489} C_VEL
LIN {X 0,Y 114.345,Z 769.234,A -85,B 0,C 180,E1 -27132.541,E2 -27132.541} C_VEL
LIN {X 0,Y 123.678,Z 764.256,A -85,B 0,C 180,E1 -27137.625,E2 -27137.625} C_VEL
LIN {X 0,Y 131.278,Z 759.393,A -85,B 0,C 180,E1 -27140.921,E2 -27140.921} C_VEL
LIN {X 0,Y 133.621,Z 757.588,A -85,B 0,C 180,E1 -27142.089,E2 -27142.089} C_VEL
LIN {X 0,Y 135.573,Z 755.835,A -85,B 0,C 180,E1 -27143.468,E2 -27143.468} C_VEL
LIN {X 0,Y 137.06,Z 754.103,A -85,B 0,C 180,E1 -27145.129,E2 -27145.129} C_VEL
LIN {X 0,Y 138.049,Z 752.335,A -85,B 0,C 180,E1 -27147.687,E2 -27147.687} C_VEL
LIN {X 0,Y 139.051,Z 749.833,A -85,B 0,C 180,E1 -27152.943,E2 -27152.943} C_VEL
LIN {X 0,Y 139.526,Z 748.883,A -85,B 0,C 180,E1 -27156.236,E2 -27156.236} C_VEL
LIN {X 0,Y 139.777,Z 748.458,A -85,B 0,C 180,E1 -27159.393,E2 -27159.393} C_VEL
LIN {X 0,Y 139.881,Z 748.549,A -85,B 0,C 180,E1 -27162.674,E2 -27162.674} C_VEL
LIN {X 0,Y 139.726,Z 749.087,A -85,B 0,C 180,E1 -27165.434,E2 -27165.434} C_VEL
LIN {X 0,Y 139.315,Z 750.13,A -85,B 0,C 180,E1 -27168.359,E2 -27168.359} C_VEL
LIN {X 0,Y 138.542,Z 751.615,A -85,B 0,C 180,E1 -27171.246,E2 -27171.246} C_VEL
LIN {X 0,Y 137.727,Z 752.675,A -85,B 0,C 180,E1 -27172.671,E2 -27172.671} C_VEL
LIN {X 0,Y 135.735,Z 754.399,A -85,B 0,C 180,E1 -27174.056,E2 -27174.056} C_VEL
LIN {X 0,Y 126.601,Z 760.288,A -85,B 0,C 180,E1 -27177.782,E2 -27177.782} C_VEL
LIN {X 0,Y 119.512,Z 764.122,A -85,B 0,C 180,E1 -27181.36,E2 -27181.36} C_VEL
LIN {X 0,Y 110.34,Z 768.085,A -85,B 0,C 180,E1 -27187.319,E2 -27187.319} C_VEL
LIN {X 0,Y 105.319,Z 769.636,A -85,B 0,C 180,E1 -27191.548,E2 -27191.548} C_VEL
LIN {X 0,Y 100.959,Z 770.57,A -85,B 0,C 180,E1 -27196.168,E2 -27196.168} C_VEL
LIN {X 0,Y 97.004,Z 770.832,A -85,B 0,C 180,E1 -27201.667,E2 -27201.667} C_VEL
LIN {X 0,Y 94.503,Z 770.709,A -85,B 0,C 180,E1 -27204.861,E2 -27204.861} C_VEL
LIN {X 0,Y 89.321,Z 769.835,A -85,B 0,C 180,E1 -27210.098,E2 -27210.098} C_VEL
LIN {X 0,Y 85.582,Z 768.595,A -85,B 0,C 180,E1 -27214.64,E2 -27214.64} C_VEL
LIN {X 0,Y 83.873,Z 767.32,A -85,B 0,C 180,E1 -27218.395,E2 -27218.395} C_VEL
LIN {X 0,Y 83.633,Z 766.795,A -85,B 0,C 180,E1 -27219.706,E2 -27219.706} C_VEL
LIN {X 0,Y 83.487,Z 763.303,A -85,B 0,C 180,E1 -27227.664,E2 -27227.664} C_VEL
LIN {X 0,Y 84.6,Z 758.138,A -85,B 0,C 180,E1 -27236.174,E2 -27236.174} C_VEL
LIN {X 0,Y 86.486,Z 752.261,A -85,B 0,C 180,E1 -27243.366,E2 -27243.366} C_VEL
LIN {X 0,Y 89.535,Z 744.66,A -85,B 0,C 180,E1 -27250.381,E2 -27250.381} C_VEL
LIN {X 0,Y 93.218,Z 736.081,A -85,B 0,C 180,E1 -27256.371,E2 -27256.371} C_VEL
LIN {X 0,Y 97.135,Z 727.056,A -85,B 0,C 180,E1 -27261.154,E2 -27261.154} C_VEL
LIN {X 0,Y 99.563,Z 721.162,A -85,B 0,C 180,E1 -27263.646,E2 -27263.646} C_VEL
LIN {X 0,Y 99.621,Z 711.781,A -85,B 0,C 180,E1 -27267.977,E2 -27267.977} C_VEL
LIN {X 0,Y 99.544,Z 707.937,A -85,B 0,C 180,E1 -27269.656,E2 -27269.656} C_VEL
LIN {X 0,Y 99.913,Z 708.496,A -85,B 0,C 180,E1 -27269.998,E2 -27269.998} C_VEL
LIN {X 0,Y 99.792,Z 718.786,A -85,B 0,C 180,E1 -27274.526,E2 -27274.526} C_VEL
LIN {X 0,Y 99.411,Z 721.092,A -85,B 0,C 180,E1 -27275.578,E2 -27275.578} C_VEL
LIN {X 0,Y 95.235,Z 731.046,A -85,B 0,C 180,E1 -27280.092,E2 -27280.092} C_VEL
LIN {X 0,Y 91.174,Z 740.177,A -85,B 0,C 180,E1 -27285.65,E2 -27285.65} C_VEL
LIN {X 0,Y 87.726,Z 748.558,A -85,B 0,C 180,E1 -27292.493,E2 -27292.493} C_VEL
LIN {X 0,Y 85.256,Z 755.129,A -85,B 0,C 180,E1 -27299.641,E2 -27299.641} C_VEL
LIN {X 0,Y 83.896,Z 759.585,A -85,B 0,C 180,E1 -27305.899,E2 -27305.899} C_VEL
LIN {X 0,Y 83.291,Z 764.401,A -85,B 0,C 180,E1 -27314.989,E2 -27314.989} C_VEL
LIN {X 0,Y 84.338,Z 767.783,A -85,B 0,C 180,E1 -27324.315,E2 -27324.315} C_VEL
LIN {X 0,Y 86.989,Z 769.615,A -85,B 0,C 180,E1 -27332.707,E2 -27332.707} C_VEL
LIN {X 0,Y 90.325,Z 770.189,A -85,B 0,C 180,E1 -27339.012,E2 -27339.012} C_VEL
LIN {X 0,Y 94.634,Z 769.979,A -85,B 0,C 180,E1 -27344.886,E2 -27344.886} C_VEL
LIN {X 0,Y 102.044,Z 768.44,A -85,B 0,C 180,E1 -27352.082,E2 -27352.082} C_VEL
LIN {X 0,Y 107.814,Z 766.522,A -85,B 0,C 180,E1 -27356.262,E2 -27356.262} C_VEL
LIN {X 0,Y 117.038,Z 762.525,A -85,B 0,C 180,E1 -27361.53,E2 -27361.53} C_VEL
LIN {X 0,Y 127.188,Z 756.847,A -85,B 0,C 180,E1 -27365.96,E2 -27365.96} C_VEL
LIN {X 0,Y 131.777,Z 753.841,A -85,B 0,C 180,E1 -27367.662,E2 -27367.662} C_VEL
LIN {X 0,Y 133.602,Z 752.271,A -85,B 0,C 180,E1 -27369.08,E2 -27369.08} C_VEL
LIN {X 0,Y 134.801,Z 750.704,A -85,B 0,C 180,E1 -27372.037,E2 -27372.037} C_VEL
LIN {X 0,Y 135.475,Z 749.571,A -85,B 0,C 180,E1 -27375.033,E2 -27375.033} C_VEL
LIN {X 0,Y 135.721,Z 749.063,A -85,B 0,C 180,E1 -27378.101,E2 -27378.101} C_VEL
LIN {X 0,Y 135.657,Z 749.081,A -85,B 0,C 180,E1 -27381.263,E2 -27381.263} C_VEL
LIN {X 0,Y 135.645,Z 749.422,A -85,B 0,C 180,E1 -27384.487,E2 -27384.487} C_VEL
LIN {X 0,Y 135.452,Z 750.378,A -85,B 0,C 180,E1 -27388.112,E2 -27388.112} C_VEL
LIN {X 0,Y 135.073,Z 751.732,A -85,B 0,C 180,E1 -27391.353,E2 -27391.353} C_VEL
LIN {X 0,Y 133.807,Z 753.119,A -85,B 0,C 180,E1 -27392.824,E2 -27392.824} C_VEL
LIN {X 0,Y 129.358,Z 756.768,A -85,B 0,C 180,E1 -27395.421,E2 -27395.421} C_VEL
LIN {X 0,Y 126.911,Z 758.542,A -85,B 0,C 180,E1 -27396.588,E2 -27396.588} C_VEL
LIN {X 0,Y 116.514,Z 764.709,A -85,B 0,C 180,E1 -27401.066,E2 -27401.066} C_VEL
LIN {X 0,Y 107.85,Z 768.823,A -85,B 0,C 180,E1 -27405.792,E2 -27405.792} C_VEL
LIN {X 0,Y 100.697,Z 771.532,A -85,B 0,C 180,E1 -27411.089,E2 -27411.089} C_VEL
LIN {X 0,Y 93.541,Z 773.359,A -85,B 0,C 180,E1 -27418.272,E2 -27418.272} C_VEL
LIN {X 0,Y 88.162,Z 773.795,A -85,B 0,C 180,E1 -27426.513,E2 -27426.513} C_VEL
LIN {X 0,Y 85.08,Z 772.819,A -85,B 0,C 180,E1 -27435.654,E2 -27435.654} C_VEL
LIN {X 0,Y 84.053,Z 770.347,A -85,B 0,C 180,E1 -27445.206,E2 -27445.206} C_VEL
LIN {X 0,Y 84.187,Z 769.084,A -85,B 0,C 180,E1 -27449.105,E2 -27449.105} C_VEL
LIN {X 0,Y 84.078,Z 771.313,A -85,B 0,C 180,E1 -27454.797,E2 -27454.797} C_VEL
LIN {X 0,Y 85.11,Z 773.827,A -85,B 0,C 180,E1 -27464.345,E2 -27464.345} C_VEL
LIN {X 0,Y 88.186,Z 774.896,A -85,B 0,C 180,E1 -27473.485,E2 -27473.485} C_VEL
LIN {X 0,Y 93.585,Z 774.542,A -85,B 0,C 180,E1 -27481.716,E2 -27481.716} C_VEL
LIN {X 0,Y 100.75,Z 772.82,A -85,B 0,C 180,E1 -27488.891,E2 -27488.891} C_VEL
LIN {X 0,Y 109.227,Z 769.678,A -85,B 0,C 180,E1 -27495.056,E2 -27495.056} C_VEL
LIN {X 0,Y 119.041,Z 764.975,A -85,B 0,C 180,E1 -27500.132,E2 -27500.132} C_VEL
LIN {X 0,Y 126.953,Z 760.355,A -85,B 0,C 180,E1 -27503.391,E2 -27503.391} C_VEL
LIN {X 0,Y 129.283,Z 758.711,A -85,B 0,C 180,E1 -27504.631,E2 -27504.631} C_VEL
LIN {X 0,Y 130.484,Z 757.641,A -85,B 0,C 180,E1 -27505.621,E2 -27505.621} C_VEL
LIN {X 0,Y 131.783,Z 756.14,A -85,B 0,C 180,E1 -27507.771,E2 -27507.771} C_VEL
LIN {X 0,Y 132.699,Z 754.38,A -85,B 0,C 180,E1 -27511.533,E2 -27511.533} C_VEL
LIN {X 0,Y 133.492,Z 753.148,A -85,B 0,C 180,E1 -27515.091,E2 -27515.091} C_VEL
LIN {X 0,Y 133.778,Z 752.592,A -85,B 0,C 180,E1 -27518.424,E2 -27518.424} C_VEL
LIN {X 0,Y 133.967,Z 752.496,A -85,B 0,C 180,E1 -27521.654,E2 -27521.654} C_VEL
LIN {X 0,Y 133.825,Z 752.876,A -85,B 0,C 180,E1 -27524.777,E2 -27524.777} C_VEL
LIN {X 0,Y 133.367,Z 753.787,A -85,B 0,C 180,E1 -27527.832,E2 -27527.832} C_VEL
LIN {X 0,Y 132.278,Z 755.174,A -85,B 0,C 180,E1 -27530.829,E2 -27530.829} C_VEL
LIN {X 0,Y 130.564,Z 756.508,A -85,B 0,C 180,E1 -27532.027,E2 -27532.027} C_VEL
LIN {X 0,Y 122.966,Z 760.985,A -85,B 0,C 180,E1 -27534.96,E2 -27534.96} C_VEL
LIN {X 0,Y 112.584,Z 765.943,A -85,B 0,C 180,E1 -27540,E2 -27540} C_VEL
LIN {X 0,Y 105.723,Z 768.48,A -85,B 0,C 180,E1 -27544.32,E2 -27544.32} C_VEL
LIN {X 0,Y 99.661,Z 770.15,A -85,B 0,C 180,E1 -27549.143,E2 -27549.143} C_VEL
LIN {X 0,Y 94.408,Z 770.98,A -85,B 0,C 180,E1 -27554.583,E2 -27554.583} C_VEL
LIN {X 0,Y 88.528,Z 770.799,A -85,B 0,C 180,E1 -27563.387,E2 -27563.387} C_VEL
LIN {X 0,Y 85.928,Z 769.845,A -85,B 0,C 180,E1 -27569.389,E2 -27569.389} C_VEL
LIN {X 0,Y 84.262,Z 768.186,A -85,B 0,C 180,E1 -27575.722,E2 -27575.722} C_VEL
LIN {X 0,Y 83.633,Z 766.795,A -85,B 0,C 180,E1 -27579.706,E2 -27579.706} C_VEL
LIN {X 0,Y 82.719,Z 765.248,A -85,B 0,C 180,E1 -27583.586,E2 -27583.586} C_VEL
LIN {X 0,Y 81.193,Z 763.395,A -85,B 0,C 180,E1 -27587.396,E2 -27587.396} C_VEL
LIN {X 0,Y 78.168,Z 757.96,A -85,B 0,C 180,E1 -27596.421,E2 -27596.421} C_VEL
LIN {X 0,Y 78.37,Z 755.14,A -85,B 0,C 180,E1 -27600.276,E2 -27600.276} C_VEL
LIN {X 0,Y 81.089,Z 747.97,A -85,B 0,C 180,E1 -27608.384,E2 -27608.384} C_VEL
LIN {X 0,Y 85.032,Z 739.319,A -85,B 0,C 180,E1 -27615.642,E2 -27615.642} C_VEL
LIN {X 0,Y 88.921,Z 730.89,A -85,B 0,C 180,E1 -27620.903,E2 -27620.903} C_VEL
LIN {X 0,Y 92.62,Z 722.521,A -85,B 0,C 180,E1 -27624.929,E2 -27624.929} C_VEL
LIN {X 0,Y 93.08,Z 719.305,A -85,B 0,C 180,E1 -27626.507,E2 -27626.507} C_VEL
LIN {X 0,Y 93.154,Z 713.005,A -85,B 0,C 180,E1 -27629.632,E2 -27629.632} C_VEL
LIN {X 0,Y 93.409,Z 713.476,A -85,B 0,C 180,E1 -27629.998,E2 -27629.998} C_VEL
LIN {X 0,Y 92.961,Z 721.211,A -85,B 0,C 180,E1 -27633.809,E2 -27633.809} C_VEL
LIN {X 0,Y 88.492,Z 731.232,A -85,B 0,C 180,E1 -27638.607,E2 -27638.607} C_VEL
LIN {X 0,Y 84.271,Z 740.286,A -85,B 0,C 180,E1 -27644.487,E2 -27644.487} C_VEL
LIN {X 0,Y 80.682,Z 748.543,A -85,B 0,C 180,E1 -27651.726,E2 -27651.726} C_VEL
LIN {X 0,Y 78.028,Z 755.346,A -85,B 0,C 180,E1 -27659.745,E2 -27659.745} C_VEL
LIN {X 0,Y 76.588,Z 760.142,A -85,B 0,C 180,E1 -27667.223,E2 -27667.223} C_VEL
LIN {X 0,Y 76.203,Z 763.863,A -85,B 0,C 180,E1 -27674.752,E2 -27674.752} C_VEL
LIN {X 0,Y 77.288,Z 767.471,A -85,B 0,C 180,E1 -27684.92,E2 -27684.92} C_VEL
LIN {X 0,Y 80.142,Z 769.542,A -85,B 0,C 180,E1 -27693.993,E2 -27693.993} C_VEL
LIN {X 0,Y 83.493,Z 770.302,A -85,B 0,C 180,E1 -27700.324,E2 -27700.324} C_VEL
LIN {X 0,Y 87.626,Z 770.398,A -85,B 0,C 180,E1 -27706.077,E2 -27706.077} C_VEL
LIN {X 0,Y 92.523,Z 769.818,A -85,B 0,C 180,E1 -27711.262,E2 -27711.262} C_VEL
LIN {X 0,Y 98.607,Z 768.49,A -85,B 0,C 180,E1 -27716.18,E2 -27716.18} C_VEL
LIN {X 0,Y 108.312,Z 765.271,A -85,B 0,C 180,E1 -27722.119,E2 -27722.119} C_VEL
LIN {X 0,Y 118.551,Z 760.62,A -85,B 0,C 180,E1 -27726.809,E2 -27726.809} C_VEL
LIN {X 0,Y 126.166,Z 756.366,A -85,B 0,C 180,E1 -27729.62,E2 -27729.62} C_VEL
LIN {X 0,Y 128.062,Z 754.975,A -85,B 0,C 180,E1 -27731.074,E2 -27731.074} C_VEL
LIN {X 0,Y 128.775,Z 754.261,A -85,B 0,C 180,E1 -27732.609,E2 -27732.609} C_VEL
LIN {X 0,Y 129.533,Z 753.324,A -85,B 0,C 180,E1 -27735.741,E2 -27735.741} C_VEL
LIN {X 0,Y 129.757,Z 752.956,A -85,B 0,C 180,E1 -27738.964,E2 -27738.964} C_VEL
LIN {X 0,Y 129.673,Z 753.167,A -85,B 0,C 180,E1 -27742.878,E2 -27742.878} C_VEL
LIN {X 0,Y 129.559,Z 753.621,A -85,B 0,C 180,E1 -27745.719,E2 -27745.719} C_VEL
LIN {X 0,Y 129.183,Z 754.764,A -85,B 0,C 180,E1 -27749.492,E2 -27749.492} C_VEL
LIN {X 0,Y 127.699,Z 756.179,A -85,B 0,C 180,E1 -27751.458,E2 -27751.458} C_VEL
LIN {X 0,Y 122.83,Z 759.537,A -85,B 0,C 180,E1 -27753.94,E2 -27753.94} C_VEL
LIN {X 0,Y 114.678,Z 764.056,A -85,B 0,C 180,E1 -27757.187,E2 -27757.187} C_VEL
LIN {X 0,Y 104.333,Z 768.67,A -85,B 0,C 180,E1 -27762.189,E2 -27762.189} C_VEL
LIN {X 0,Y 95.278,Z 771.686,A -85,B 0,C 180,E1 -27768.407,E2 -27768.407} C_VEL
LIN {X 0,Y 87.581,Z 773.303,A -85,B 0,C 180,E1 -27775.828,E2 -27775.828} C_VEL
LIN {X 0,Y 81.675,Z 773.513,A -85,B 0,C 180,E1 -27784.519,E2 -27784.519} C_VEL
LIN {X 0,Y 78.203,Z 772.303,A -85,B 0,C 180,E1 -27794.362,E2 -27794.362} C_VEL
LIN {X 0,Y 77.002,Z 769.655,A -85,B 0,C 180,E1 -27804.766,E2 -27804.766} C_VEL
LIN {X 0,Y 77.148,Z 768.17,A -85,B 0,C 180,E1 -27809.024,E2 -27809.024} C_VEL
LIN {X 0,Y 77.026,Z 770.586,A -85,B 0,C 180,E1 -27815.237,E2 -27815.237} C_VEL
LIN {X 0,Y 78.259,Z 773.291,A -85,B 0,C 180,E1 -27825.632,E2 -27825.632} C_VEL
LIN {X 0,Y 81.701,Z 774.557,A -85,B 0,C 180,E1 -27835.476,E2 -27835.476} C_VEL
LIN {X 0,Y 87.623,Z 774.471,A -85,B 0,C 180,E1 -27844.158,E2 -27844.158} C_VEL
LIN {X 0,Y 95.33,Z 772.958,A -85,B 0,C 180,E1 -27851.57,E2 -27851.57} C_VEL
LIN {X 0,Y 104.345,Z 770.076,A -85,B 0,C 180,E1 -27857.809,E2 -27857.809} C_VEL
LIN {X 0,Y 114.654,Z 765.69,A -85,B 0,C 180,E1 -27862.834,E2 -27862.834} C_VEL
LIN {X 0,Y 122.839,Z 761.348,A -85,B 0,C 180,E1 -27866.058,E2 -27866.058} C_VEL
LIN {X 0,Y 124.992,Z 759.841,A -85,B 0,C 180,E1 -27867.504,E2 -27867.504} C_VEL
LIN {X 0,Y 126.038,Z 758.643,A -85,B 0,C 180,E1 -27869.878,E2 -27869.878} C_VEL
LIN {X 0,Y 127.011,Z 757.245,A -85,B 0,C 180,E1 -27873.726,E2 -27873.726} C_VEL
LIN {X 0,Y 127.542,Z 756.467,A -85,B 0,C 180,E1 -27877.311,E2 -27877.311} C_VEL
LIN {X 0,Y 127.834,Z 756.189,A -85,B 0,C 180,E1 -27880.74,E2 -27880.74} C_VEL
LIN {X 0,Y 127.728,Z 756.419,A -85,B 0,C 180,E1 -27884.031,E2 -27884.031} C_VEL
LIN {X 0,Y 127.237,Z 757.158,A -85,B 0,C 180,E1 -27887.236,E2 -27887.236} C_VEL
LIN {X 0,Y 126.61,Z 757.76,A -85,B 0,C 180,E1 -27888.797,E2 -27888.797} C_VEL
LIN {X 0,Y 124.341,Z 759.204,A -85,B 0,C 180,E1 -27890.237,E2 -27890.237} C_VEL
LIN {X 0,Y 112.916,Z 764.789,A -85,B 0,C 180,E1 -27894.794,E2 -27894.794} C_VEL
LIN {X 0,Y 103.138,Z 768.417,A -85,B 0,C 180,E1 -27900,E2 -27900} C_VEL
LIN {X 0,Y 97.078,Z 770.016,A -85,B 0,C 180,E1 -27904.152,E2 -27904.152} C_VEL
LIN {X 0,Y 91.585,Z 771.017,A -85,B 0,C 180,E1 -27908.829,E2 -27908.829} C_VEL
LIN {X 0,Y 86.884,Z 771.342,A -85,B 0,C 180,E1 -27914.044,E2 -27914.044} C_VEL
LIN {X 0,Y 82.549,Z 770.987,A -85,B 0,C 180,E1 -27920.521,E2 -27920.521} C_VEL
LIN {X 0,Y 79.269,Z 769.867,A -85,B 0,C 180,E1 -27927.547,E2 -27927.547} C_VEL
LIN {X 0,Y 77.236,Z 767.939,A -85,B 0,C 180,E1 -27935.018,E2 -27935.018} C_VEL
LIN {X 0,Y 76.307,Z 764.273,A -85,B 0,C 180,E1 -27944.772,E2 -27944.772} C_VEL
LIN {X 0,Y 76.884,Z 760.205,A -85,B 0,C 180,E1 -27952.705,E2 -27952.705} C_VEL
LIN {X 0,Y 78.37,Z 755.14,A -85,B 0,C 180,E1 -27960.276,E2 -27960.276} C_VEL
LIN {X 0,Y 78.769,Z 752.193,A -85,B 0,C 180,E1 -27963.954,E2 -27963.954} C_VEL
LIN {X 0,Y 78.199,Z 746.796,A -85,B 0,C 180,E1 -27969.994,E2 -27969.994} C_VEL
LIN {X 0,Y 78.198,Z 740.743,A -85,B 0,C 180,E1 -27975.83,E2 -27975.83} C_VEL
LIN {X 0,Y 79.45,Z 736.76,A -85,B 0,C 180,E1 -27978.96,E2 -27978.96} C_VEL
LIN {X 0,Y 83.959,Z 727.438,A -85,B 0,C 180,E1 -27984.594,E2 -27984.594} C_VEL
LIN {X 0,Y 86.319,Z 722.212,A -85,B 0,C 180,E1 -27987.099,E2 -27987.099} C_VEL
LIN {X 0,Y 86.7,Z 717.642,A -85,B 0,C 180,E1 -27989.708,E2 -27989.708} C_VEL
LIN {X 0,Y 86.567,Z 721.253,A -85,B 0,C 180,E1 -27991.743,E2 -27991.743} C_VEL
LIN {X 0,Y 81.909,Z 731.225,A -85,B 0,C 180,E1 -27996.773,E2 -27996.773} C_VEL
LIN {X 0,Y 78.086,Z 738.989,A -85,B 0,C 180,E1 -28002.001,E2 -28002.001} C_VEL
LIN {X 0,Y 74.387,Z 746.917,A -85,B 0,C 180,E1 -28009.127,E2 -28009.127} C_VEL
LIN {X 0,Y 71.373,Z 753.923,A -85,B 0,C 180,E1 -28017.597,E2 -28017.597} C_VEL
LIN {X 0,Y 69.615,Z 759.233,A -85,B 0,C 180,E1 -28026.133,E2 -28026.133} C_VEL
LIN {X 0,Y 69.128,Z 763.582,A -85,B 0,C 180,E1 -28035.366,E2 -28035.366} C_VEL
LIN {X 0,Y 69.858,Z 766.502,A -85,B 0,C 180,E1 -28043.59,E2 -28043.59} C_VEL
LIN {X 0,Y 71.863,Z 768.648,A -85,B 0,C 180,E1 -28051.658,E2 -28051.658} C_VEL
LIN {X 0,Y 75.158,Z 770.038,A -85,B 0,C 180,E1 -28059.236,E2 -28059.236} C_VEL
LIN {X 0,Y 79.62,Z 770.629,A -85,B 0,C 180,E1 -28066.148,E2 -28066.148} C_VEL
LIN {X 0,Y 85.092,Z 770.456,A -85,B 0,C 180,E1 -28072.338,E2 -28072.338} C_VEL
LIN {X 0,Y 94.872,Z 768.79,A -85,B 0,C 180,E1 -28080,E2 -28080} C_VEL
LIN {X 0,Y 101.705,Z 766.845,A -85,B 0,C 180,E1 -28083.962,E2 -28083.962} C_VEL
LIN {X 0,Y 111.717,Z 763.061,A -85,B 0,C 180,E1 -28088.546,E2 -28088.546} C_VEL
LIN {X 0,Y 120.665,Z 758.724,A -85,B 0,C 180,E1 -28091.762,E2 -28091.762} C_VEL
LIN {X 0,Y 122.604,Z 757.512,A -85,B 0,C 180,E1 -28093.255,E2 -28093.255} C_VEL
LIN {X 0,Y 123.411,Z 756.784,A -85,B 0,C 180,E1 -28096.543,E2 -28096.543} C_VEL
LIN {X 0,Y 123.559,Z 756.589,A -85,B 0,C 180,E1 -28099.955,E2 -28099.955} C_VEL
LIN {X 0,Y 123.451,Z 756.977,A -85,B 0,C 180,E1 -28104.378,E2 -28104.378} C_VEL
LIN {X 0,Y 123.147,Z 757.597,A -85,B 0,C 180,E1 -28107.165,E2 -28107.165} C_VEL
LIN {X 0,Y 121.6,Z 758.967,A -85,B 0,C 180,E1 -28109.898,E2 -28109.898} C_VEL
LIN {X 0,Y 119.017,Z 760.527,A -85,B 0,C 180,E1 -28111.107,E2 -28111.107} C_VEL
LIN {X 0,Y 110.558,Z 764.794,A -85,B 0,C 180,E1 -28114.273,E2 -28114.273} C_VEL
LIN {X 0,Y 99.718,Z 769.058,A -85,B 0,C 180,E1 -28119.174,E2 -28119.174} C_VEL
LIN {X 0,Y 90.096,Z 771.842,A -85,B 0,C 180,E1 -28125.411,E2 -28125.411} C_VEL
LIN {X 0,Y 81.791,Z 773.21,A -85,B 0,C 180,E1 -28133.027,E2 -28133.027} C_VEL
LIN {X 0,Y 75.308,Z 773.169,A -85,B 0,C 180,E1 -28142.188,E2 -28142.188} C_VEL
LIN {X 0,Y 71.377,Z 771.769,A -85,B 0,C 180,E1 -28152.822,E2 -28152.822} C_VEL
LIN {X 0,Y 70.381,Z 770.527,A -85,B 0,C 180,E1 -28158.482,E2 -28158.482} C_VEL
LIN {X 0,Y 70.113,Z 767.33,A -85,B 0,C 180,E1 -28169.105,E2 -28169.105} C_VEL
LIN {X 0,Y 69.99,Z 769.774,A -85,B 0,C 180,E1 -28175.765,E2 -28175.765} C_VEL
LIN {X 0,Y 71.459,Z 772.728,A -85,B 0,C 180,E1 -28187.163,E2 -28187.163} C_VEL
LIN {X 0,Y 75.335,Z 774.193,A -85,B 0,C 180,E1 -28197.806,E2 -28197.806} C_VEL
LIN {X 0,Y 81.845,Z 774.317,A -85,B 0,C 180,E1 -28206.95,E2 -28206.95} C_VEL
LIN {X 0,Y 90.145,Z 773.094,A -85,B 0,C 180,E1 -28214.563,E2 -28214.563} C_VEL
LIN {X 0,Y 99.726,Z 770.451,A -85,B 0,C 180,E1 -28220.826,E2 -28220.826} C_VEL
LIN {X 0,Y 110.543,Z 766.356,A -85,B 0,C 180,E1 -28225.743,E2 -28225.743} C_VEL
LIN {X 0,Y 116.217,Z 763.737,A -85,B 0,C 180,E1 -28227.849,E2 -28227.849} C_VEL
LIN {X 0,Y 118.878,Z 762.304,A -85,B 0,C 180,E1 -28229.01,E2 -28229.01} C_VEL
LIN {X 0,Y 120.139,Z 761.077,A -85,B 0,C 180,E1 -28232.096,E2 -28232.096} C_VEL
LIN {X 0,Y 121.005,Z 760.093,A -85,B 0,C 180,E1 -28236.011,E2 -28236.011} C_VEL
LIN {X 0,Y 121.519,Z 759.585,A -85,B 0,C 180,E1 -28239.696,E2 -28239.696} C_VEL
LIN {X 0,Y 121.452,Z 759.686,A -85,B 0,C 180,E1 -28243.182,E2 -28243.182} C_VEL
LIN {X 0,Y 120.957,Z 760.208,A -85,B 0,C 180,E1 -28246.561,E2 -28246.561} C_VEL
LIN {X 0,Y 118.885,Z 761.35,A -85,B 0,C 180,E1 -28248.059,E2 -28248.059} C_VEL
LIN {X 0,Y 107.347,Z 766.278,A -85,B 0,C 180,E1 -28252.476,E2 -28252.476} C_VEL
LIN {X 0,Y 98.534,Z 769.068,A -85,B 0,C 180,E1 -28256.945,E2 -28256.945} C_VEL
LIN {X 0,Y 91.402,Z 770.685,A -85,B 0,C 180,E1 -28261.591,E2 -28261.591} C_VEL
LIN {X 0,Y 84.973,Z 771.48,A -85,B 0,C 180,E1 -28267.004,E2 -28267.004} C_VEL
LIN {X 0,Y 77.716,Z 771.344,A -85,B 0,C 180,E1 -28275.742,E2 -28275.742} C_VEL
LIN {X 0,Y 74.059,Z 770.437,A -85,B 0,C 180,E1 -28282.308,E2 -28282.308} C_VEL
